LIN {X 0,Y 547.028,Z 596.722,A -85,B 0,C 180,E1 3579.172,E2 3579.172} C_VEL
LIN {X 0,Y 546.524,Z 623.669,A -85,B 0,C 180,E1 3580.328,E2 3580.328} C_VEL
LIN {X 0,Y 545.905,Z 649.048,A -85,B 0,C 180,E1 3582.094,E2 3582.094} C_VEL
LIN {X 0,Y 545.325,Z 670.672,A -85,B 0,C 180,E1 3584.351,E2 3584.351} C_VEL
LIN {X 0,Y 545.02,Z 688.06,A -85,B 0,C 180,E1 3587.017,E2 3587.017} C_VEL
LIN {X 0,Y 544.801,Z 699.894,A -85,B 0,C 180,E1 3589.924,E2 3589.924} C_VEL
LIN {X 0,Y 544.735,Z 704.998,A -85,B 0,C 180,E1 3592.042,E2 3592.042} C_VEL
LIN {X 0,Y 544.721,Z 707.404,A -85,B 0,C 180,E1 3595.236,E2 3595.236} C_VEL
LIN {X 0,Y 544.817,Z 705.335,A -85,B 0,C 180,E1 3597.622,E2 3597.622} C_VEL
LIN {X 0,Y 544.899,Z 697.263,A -85,B 0,C 180,E1 3600.797,E2 3600.797} C_VEL
LIN {X 0,Y 545.082,Z 683.494,A -85,B 0,C 180,E1 3603.697,E2 3603.697} C_VEL
LIN {X 0,Y 545.462,Z 664.993,A -85,B 0,C 180,E1 3606.247,E2 3606.247} C_VEL
LIN {X 0,Y 546.119,Z 641.134,A -85,B 0,C 180,E1 3608.445,E2 3608.445} C_VEL
LIN {X 0,Y 546.671,Z 615.982,A -85,B 0,C 180,E1 3609.983,E2 3609.983} C_VEL
LIN {X 0,Y 547.21,Z 587.354,A -85,B 0,C 180,E1 3611.001,E2 3611.001} C_VEL
LIN {X 0,Y 546.153,Z 557.095,A -85,B 0,C 180,E1 3611.528,E2 3611.528} C_VEL
LIN {X 0,Y 544.539,Z 549.53,A -85,B 0,C 180,E1 3611.757,E2 3611.757} C_VEL
LIN {X 0,Y 544.29,Z 549.53,A -85,B 0,C 180,E1 3617.76,E2 3617.76} C_VEL
LIN {X 0,Y 544.118,Z 549.53,A -85,B 0,C 180,E1 3623.753,E2 3623.753} C_VEL
LIN {X 0,Y 543.994,Z 549.53,A -85,B 0,C 180,E1 3629.959,E2 3629.959} C_VEL
LIN {X 0,Y 543.92,Z 549.53,A -85,B 0,C 180,E1 3635.639,E2 3635.639} C_VEL
LIN {X 0,Y 543.965,Z 549.53,A -85,B 0,C 180,E1 3641.748,E2 3641.748} C_VEL
LIN {X 0,Y 544.059,Z 549.53,A -85,B 0,C 180,E1 3648.261,E2 3648.261} C_VEL
LIN {X 0,Y 543.981,Z 549.53,A -85,B 0,C 180,E1 3654.366,E2 3654.366} C_VEL
LIN {X 0,Y 543.974,Z 549.53,A -85,B 0,C 180,E1 3660.041,E2 3660.041} C_VEL
LIN {X 0,Y 544.383,Z 549.53,A -85,B 0,C 180,E1 3664.815,E2 3664.815} C_VEL
LIN {X 0,Y 551.536,Z 570.193,A -85,B 0,C 180,E1 3665.614,E2 3665.614} C_VEL
LIN {X 0,Y 550.555,Z 607.701,A -85,B 0,C 180,E1 3666.786,E2 3666.786} C_VEL
LIN {X 0,Y 549.229,Z 644.248,A -85,B 0,C 180,E1 3668.649,E2 3668.649} C_VEL
LIN {X 0,Y 547.877,Z 676.541,A -85,B 0,C 180,E1 3670.994,E2 3670.994} C_VEL
LIN {X 0,Y 546.564,Z 706.625,A -85,B 0,C 180,E1 3673.971,E2 3673.971} C_VEL
LIN {X 0,Y 545.565,Z 730.848,A -85,B 0,C 180,E1 3677.215,E2 3677.215} C_VEL
LIN {X 0,Y 545.084,Z 748.889,A -85,B 0,C 180,E1 3680.438,E2 3680.438} C_VEL
LIN {X 0,Y 544.734,Z 763.268,A -85,B 0,C 180,E1 3684.037,E2 3684.037} C_VEL
LIN {X 0,Y 544.715,Z 772.438,A -85,B 0,C 180,E1 3687.618,E2 3687.618} C_VEL
LIN {X 0,Y 544.588,Z 777.144,A -85,B 0,C 180,E1 3691.588,E2 3691.588} C_VEL
LIN {X 0,Y 544.66,Z 776.874,A -85,B 0,C 180,E1 3694.769,E2 3694.769} C_VEL
LIN {X 0,Y 544.677,Z 771.522,A -85,B 0,C 180,E1 3698.766,E2 3698.766} C_VEL
LIN {X 0,Y 544.773,Z 761.522,A -85,B 0,C 180,E1 3702.398,E2 3702.398} C_VEL
LIN {X 0,Y 545.169,Z 745.947,A -85,B 0,C 180,E1 3706.071,E2 3706.071} C_VEL
LIN {X 0,Y 545.847,Z 724.204,A -85,B 0,C 180,E1 3709.682,E2 3709.682} C_VEL
LIN {X 0,Y 546.935,Z 698.541,A -85,B 0,C 180,E1 3712.832,E2 3712.832} C_VEL
LIN {X 0,Y 548.289,Z 666.942,A -85,B 0,C 180,E1 3715.697,E2 3715.697} C_VEL
LIN {X 0,Y 549.53,Z 634.518,A -85,B 0,C 180,E1 3717.832,E2 3717.832} C_VEL
LIN {X 0,Y 550.827,Z 598.514,A -85,B 0,C 180,E1 3719.477,E2 3719.477} C_VEL
LIN {X 0,Y 550.795,Z 568.148,A -85,B 0,C 180,E1 3720.384,E2 3720.384} C_VEL
LIN {X 0,Y 544.129,Z 549.53,A -85,B 0,C 180,E1 3721.134,E2 3721.134} C_VEL
LIN {X 0,Y 544.13,Z 549.53,A -85,B 0,C 180,E1 3726.456,E2 3726.456} C_VEL
LIN {X 0,Y 544.008,Z 549.53,A -85,B 0,C 180,E1 3731.744,E2 3731.744} C_VEL
LIN {X 0,Y 544.033,Z 549.53,A -85,B 0,C 180,E1 3738.504,E2 3738.504} C_VEL
LIN {X 0,Y 544.169,Z 549.53,A -85,B 0,C 180,E1 3744.38,E2 3744.38} C_VEL
LIN {X 0,Y 544.074,Z 549.53,A -85,B 0,C 180,E1 3750.046,E2 3750.046} C_VEL
LIN {X 0,Y 544.017,Z 549.53,A -85,B 0,C 180,E1 3756.273,E2 3756.273} C_VEL
LIN {X 0,Y 544.219,Z 549.53,A -85,B 0,C 180,E1 3761.604,E2 3761.604} C_VEL
LIN {X 0,Y 546.614,Z 578.067,A -85,B 0,C 180,E1 3762.063,E2 3762.063} C_VEL
LIN {X 0,Y 546.452,Z 611.547,A -85,B 0,C 180,E1 3762.642,E2 3762.642} C_VEL
LIN {X 0,Y 546.062,Z 638.227,A -85,B 0,C 180,E1 3763.751,E2 3763.751} C_VEL
LIN {X 0,Y 545.544,Z 661.449,A -85,B 0,C 180,E1 3765.432,E2 3765.432} C_VEL
LIN {X 0,Y 545.125,Z 679.302,A -85,B 0,C 180,E1 3767.405,E2 3767.405} C_VEL
LIN {X 0,Y 544.917,Z 694.025,A -85,B 0,C 180,E1 3769.891,E2 3769.891} C_VEL
LIN {X 0,Y 544.794,Z 703.355,A -85,B 0,C 180,E1 3772.538,E2 3772.538} C_VEL
LIN {X 0,Y 544.727,Z 707.246,A -85,B 0,C 180,E1 3775.229,E2 3775.229} C_VEL
LIN {X 0,Y 544.711,Z 707.192,A -85,B 0,C 180,E1 3776.82,E2 3776.82} C_VEL
LIN {X 0,Y 544.857,Z 702.766,A -85,B 0,C 180,E1 3779.6,E2 3779.6} C_VEL
LIN {X 0,Y 544.936,Z 692.366,A -85,B 0,C 180,E1 3782.377,E2 3782.377} C_VEL
LIN {X 0,Y 545.244,Z 676.093,A -85,B 0,C 180,E1 3784.92,E2 3784.92} C_VEL
LIN {X 0,Y 545.685,Z 656.173,A -85,B 0,C 180,E1 3786.945,E2 3786.945} C_VEL
LIN {X 0,Y 546.186,Z 633.014,A -85,B 0,C 180,E1 3788.436,E2 3788.436} C_VEL
LIN {X 0,Y 546.479,Z 607.222,A -85,B 0,C 180,E1 3789.383,E2 3789.383} C_VEL
LIN {X 0,Y 545.692,Z 554.823,A -85,B 0,C 180,E1 3790.17,E2 3790.17} C_VEL
LIN {X 0,Y 544.581,Z 549.53,A -85,B 0,C 180,E1 3790.348,E2 3790.348} C_VEL
LIN {X 0,Y 544.209,Z 549.53,A -85,B 0,C 180,E1 3792.982,E2 3792.982} C_VEL
LIN {X 0,Y 540.252,Z 549.53,A -85,B 0,C 180,E1 3794.779,E2 3794.779} C_VEL
LIN {X 0,Y 536.278,Z 549.53,A -85,B 0,C 180,E1 3796.602,E2 3796.602} C_VEL
LIN {X 0,Y 536.17,Z 549.53,A -85,B 0,C 180,E1 3801.741,E2 3801.741} C_VEL
LIN {X 0,Y 536.063,Z 549.53,A -85,B 0,C 180,E1 3806.765,E2 3806.765} C_VEL
LIN {X 0,Y 535.986,Z 549.53,A -85,B 0,C 180,E1 3812.358,E2 3812.358} C_VEL
LIN {X 0,Y 536.152,Z 549.53,A -85,B 0,C 180,E1 3818.253,E2 3818.253} C_VEL
LIN {X 0,Y 536.007,Z 549.53,A -85,B 0,C 180,E1 3824.73,E2 3824.73} C_VEL
LIN {X 0,Y 535.97,Z 549.53,A -85,B 0,C 180,E1 3829.636,E2 3829.636} C_VEL
LIN {X 0,Y 536.088,Z 550.016,A -85,B 0,C 180,E1 3835.356,E2 3835.356} C_VEL
LIN {X 0,Y 537.029,Z 553.098,A -85,B 0,C 180,E1 3836.078,E2 3836.078} C_VEL
LIN {X 0,Y 547.19,Z 573.958,A -85,B 0,C 180,E1 3837.11,E2 3837.11} C_VEL
LIN {X 0,Y 546.77,Z 626.968,A -85,B 0,C 180,E1 3838.085,E2 3838.085} C_VEL
LIN {X 0,Y 545.503,Z 664.523,A -85,B 0,C 180,E1 3839.384,E2 3839.384} C_VEL
LIN {X 0,Y 543.745,Z 701.396,A -85,B 0,C 180,E1 3841.3,E2 3841.3} C_VEL
LIN {X 0,Y 541.756,Z 736.91,A -85,B 0,C 180,E1 3843.864,E2 3843.864} C_VEL
LIN {X 0,Y 539.937,Z 768.966,A -85,B 0,C 180,E1 3846.963,E2 3846.963} C_VEL
LIN {X 0,Y 538.457,Z 797.181,A -85,B 0,C 180,E1 3850.559,E2 3850.559} C_VEL
LIN {X 0,Y 537.455,Z 819.461,A -85,B 0,C 180,E1 3854.319,E2 3854.319} C_VEL
LIN {X 0,Y 536.952,Z 836.542,A -85,B 0,C 180,E1 3858.242,E2 3858.242} C_VEL
LIN {X 0,Y 536.771,Z 847.704,A -85,B 0,C 180,E1 3861.918,E2 3861.918} C_VEL
LIN {X 0,Y 536.661,Z 853.979,A -85,B 0,C 180,E1 3865.16,E2 3865.16} C_VEL
LIN {X 0,Y 536.666,Z 857.105,A -85,B 0,C 180,E1 3868.388,E2 3868.388} C_VEL
LIN {X 0,Y 536.801,Z 857.105,A -85,B 0,C 180,E1 3871.611,E2 3871.611} C_VEL
LIN {X 0,Y 536.76,Z 852.747,A -85,B 0,C 180,E1 3875.647,E2 3875.647} C_VEL
LIN {X 0,Y 536.826,Z 843.325,A -85,B 0,C 180,E1 3879.711,E2 3879.711} C_VEL
LIN {X 0,Y 537.257,Z 827.755,A -85,B 0,C 180,E1 3883.938,E2 3883.938} C_VEL
LIN {X 0,Y 538.05,Z 806.656,A -85,B 0,C 180,E1 3887.971,E2 3887.971} C_VEL
LIN {X 0,Y 539.341,Z 780.531,A -85,B 0,C 180,E1 3891.684,E2 3891.684} C_VEL
LIN {X 0,Y 541.056,Z 749.2,A -85,B 0,C 180,E1 3895.049,E2 3895.049} C_VEL
LIN {X 0,Y 543.025,Z 714.333,A -85,B 0,C 180,E1 3897.86,E2 3897.86} C_VEL
LIN {X 0,Y 544.929,Z 676.974,A -85,B 0,C 180,E1 3900.05,E2 3900.05} C_VEL
LIN {X 0,Y 546.442,Z 637.3,A -85,B 0,C 180,E1 3901.622,E2 3901.622} C_VEL
LIN {X 0,Y 547.443,Z 597.917,A -85,B 0,C 180,E1 3902.505,E2 3902.505} C_VEL
LIN {X 0,Y 546.759,Z 573.274,A -85,B 0,C 180,E1 3902.929,E2 3902.929} C_VEL
LIN {X 0,Y 536.066,Z 549.77,A -85,B 0,C 180,E1 3904.094,E2 3904.094} C_VEL
LIN {X 0,Y 536.186,Z 549.53,A -85,B 0,C 180,E1 3908.259,E2 3908.259} C_VEL
LIN {X 0,Y 535.987,Z 549.53,A -85,B 0,C 180,E1 3914.742,E2 3914.742} C_VEL
LIN {X 0,Y 536.086,Z 549.53,A -85,B 0,C 180,E1 3919.657,E2 3919.657} C_VEL
LIN {X 0,Y 536.037,Z 549.53,A -85,B 0,C 180,E1 3924.733,E2 3924.733} C_VEL
LIN {X 0,Y 536.049,Z 549.53,A -85,B 0,C 180,E1 3930.781,E2 3930.781} C_VEL
LIN {X 0,Y 536.168,Z 549.53,A -85,B 0,C 180,E1 3936.799,E2 3936.799} C_VEL
LIN {X 0,Y 536.352,Z 549.882,A -85,B 0,C 180,E1 3938.06,E2 3938.06} C_VEL
LIN {X 0,Y 539.4,Z 567.141,A -85,B 0,C 180,E1 3938.367,E2 3938.367} C_VEL
LIN {X 0,Y 539.351,Z 599.199,A -85,B 0,C 180,E1 3939.037,E2 3939.037} C_VEL
LIN {X 0,Y 538.815,Z 627.007,A -85,B 0,C 180,E1 3940.276,E2 3940.276} C_VEL
LIN {X 0,Y 538.193,Z 651.43,A -85,B 0,C 180,E1 3942.039,E2 3942.039} C_VEL
LIN {X 0,Y 537.578,Z 672.435,A -85,B 0,C 180,E1 3944.329,E2 3944.329} C_VEL
LIN {X 0,Y 537.147,Z 688.92,A -85,B 0,C 180,E1 3947.016,E2 3947.016} C_VEL
LIN {X 0,Y 536.867,Z 701.196,A -85,B 0,C 180,E1 3950.294,E2 3950.294} C_VEL
LIN {X 0,Y 536.836,Z 704.882,A -85,B 0,C 180,E1 3951.924,E2 3951.924} C_VEL
LIN {X 0,Y 536.812,Z 707.4,A -85,B 0,C 180,E1 3955.166,E2 3955.166} C_VEL
LIN {X 0,Y 536.855,Z 704.123,A -85,B 0,C 180,E1 3958.393,E2 3958.393} C_VEL
LIN {X 0,Y 536.903,Z 694.456,A -85,B 0,C 180,E1 3961.614,E2 3961.614} C_VEL
LIN {X 0,Y 537.262,Z 681.227,A -85,B 0,C 180,E1 3964.279,E2 3964.279} C_VEL
LIN {X 0,Y 537.883,Z 661.608,A -85,B 0,C 180,E1 3966.852,E2 3966.852} C_VEL
LIN {X 0,Y 538.498,Z 638.728,A -85,B 0,C 180,E1 3968.87,E2 3968.87} C_VEL
LIN {X 0,Y 539.16,Z 612.131,A -85,B 0,C 180,E1 3970.384,E2 3970.384} C_VEL
LIN {X 0,Y 539.616,Z 584.105,A -85,B 0,C 180,E1 3971.293,E2 3971.293} C_VEL
LIN {X 0,Y 538.584,Z 558.624,A -85,B 0,C 180,E1 3971.715,E2 3971.715} C_VEL
LIN {X 0,Y 536.63,Z 549.53,A -85,B 0,C 180,E1 3971.902,E2 3971.902} C_VEL
LIN {X 0,Y 536.36,Z 549.53,A -85,B 0,C 180,E1 3978.032,E2 3978.032} C_VEL
LIN {X 0,Y 536.24,Z 549.53,A -85,B 0,C 180,E1 3983.206,E2 3983.206} C_VEL
LIN {X 0,Y 536.062,Z 549.53,A -85,B 0,C 180,E1 3989.221,E2 3989.221} C_VEL
LIN {X 0,Y 536.025,Z 549.53,A -85,B 0,C 180,E1 3994.271,E2 3994.271} C_VEL
LIN {X 0,Y 535.971,Z 549.53,A -85,B 0,C 180,E1 4000.513,E2 4000.513} C_VEL
LIN {X 0,Y 536.049,Z 549.53,A -85,B 0,C 180,E1 4007.053,E2 4007.053} C_VEL
LIN {X 0,Y 536.15,Z 549.53,A -85,B 0,C 180,E1 4012.012,E2 4012.012} C_VEL
LIN {X 0,Y 536.009,Z 549.53,A -85,B 0,C 180,E1 4017.659,E2 4017.659} C_VEL
LIN {X 0,Y 536.434,Z 549.53,A -85,B 0,C 180,E1 4024.363,E2 4024.363} C_VEL
LIN {X 0,Y 544.5,Z 571.697,A -85,B 0,C 180,E1 4025.269,E2 4025.269} C_VEL
LIN {X 0,Y 543.373,Z 608.888,A -85,B 0,C 180,E1 4026.466,E2 4026.466} C_VEL
LIN {X 0,Y 541.907,Z 644.984,A -85,B 0,C 180,E1 4028.346,E2 4028.346} C_VEL
LIN {X 0,Y 540.436,Z 676.308,A -85,B 0,C 180,E1 4030.655,E2 4030.655} C_VEL
LIN {X 0,Y 538.983,Z 705.238,A -85,B 0,C 180,E1 4033.531,E2 4033.531} C_VEL
LIN {X 0,Y 537.85,Z 729.819,A -85,B 0,C 180,E1 4036.822,E2 4036.822} C_VEL
LIN {X 0,Y 537.262,Z 749.105,A -85,B 0,C 180,E1 4040.297,E2 4040.297} C_VEL
LIN {X 0,Y 536.857,Z 763.401,A -85,B 0,C 180,E1 4043.949,E2 4043.949} C_VEL
LIN {X 0,Y 536.833,Z 772.522,A -85,B 0,C 180,E1 4047.583,E2 4047.583} C_VEL
LIN {X 0,Y 536.698,Z 777.155,A -85,B 0,C 180,E1 4051.612,E2 4051.612} C_VEL
LIN {X 0,Y 536.752,Z 776.846,A -85,B 0,C 180,E1 4054.839,E2 4054.839} C_VEL
LIN {X 0,Y 536.791,Z 771.439,A -85,B 0,C 180,E1 4058.896,E2 4058.896} C_VEL
LIN {X 0,Y 536.909,Z 761.358,A -85,B 0,C 180,E1 4062.583,E2 4062.583} C_VEL
LIN {X 0,Y 537.478,Z 744.404,A -85,B 0,C 180,E1 4066.568,E2 4066.568} C_VEL
LIN {X 0,Y 538.324,Z 721.745,A -85,B 0,C 180,E1 4070.279,E2 4070.279} C_VEL
LIN {X 0,Y 539.492,Z 694.967,A -85,B 0,C 180,E1 4073.493,E2 4073.493} C_VEL
LIN {X 0,Y 540.953,Z 665.008,A -85,B 0,C 180,E1 4076.177,E2 4076.177} C_VEL
LIN {X 0,Y 542.504,Z 629.524,A -85,B 0,C 180,E1 4078.465,E2 4078.465} C_VEL
LIN {X 0,Y 543.811,Z 593.165,A -85,B 0,C 180,E1 4080.033,E2 4080.033} C_VEL
LIN {X 0,Y 543.789,Z 570.399,A -85,B 0,C 180,E1 4080.716,E2 4080.716} C_VEL
LIN {X 0,Y 536.243,Z 549.53,A -85,B 0,C 180,E1 4081.594,E2 4081.594} C_VEL
LIN {X 0,Y 536.225,Z 549.53,A -85,B 0,C 180,E1 4086.231,E2 4086.231} C_VEL
LIN {X 0,Y 535.988,Z 549.53,A -85,B 0,C 180,E1 4092.514,E2 4092.514} C_VEL
LIN {X 0,Y 536.002,Z 549.53,A -85,B 0,C 180,E1 4097.488,E2 4097.488} C_VEL
LIN {X 0,Y 536.248,Z 549.53,A -85,B 0,C 180,E1 4103.771,E2 4103.771} C_VEL
LIN {X 0,Y 536.183,Z 549.53,A -85,B 0,C 180,E1 4109.559,E2 4109.559} C_VEL
LIN {X 0,Y 536.048,Z 549.53,A -85,B 0,C 180,E1 4115.018,E2 4115.018} C_VEL
LIN {X 0,Y 536.304,Z 549.53,A -85,B 0,C 180,E1 4121.416,E2 4121.416} C_VEL
LIN {X 0,Y 538.926,Z 577.898,A -85,B 0,C 180,E1 4121.874,E2 4121.874} C_VEL
LIN {X 0,Y 538.796,Z 613.16,A -85,B 0,C 180,E1 4122.493,E2 4122.493} C_VEL
LIN {X 0,Y 538.407,Z 638.091,A -85,B 0,C 180,E1 4123.531,E2 4123.531} C_VEL
LIN {X 0,Y 537.887,Z 661.122,A -85,B 0,C 180,E1 4125.163,E2 4125.163} C_VEL
LIN {X 0,Y 537.428,Z 679.88,A -85,B 0,C 180,E1 4127.221,E2 4127.221} C_VEL
LIN {X 0,Y 537.121,Z 694.712,A -85,B 0,C 180,E1 4129.759,E2 4129.759} C_VEL
LIN {X 0,Y 536.956,Z 704.116,A -85,B 0,C 180,E1 4132.536,E2 4132.536} C_VEL
LIN {X 0,Y 536.848,Z 707.814,A -85,B 0,C 180,E1 4135.159,E2 4135.159} C_VEL
LIN {X 0,Y 536.839,Z 707.82,A -85,B 0,C 180,E1 4136.773,E2 4136.773} C_VEL
LIN {X 0,Y 537.025,Z 703.659,A -85,B 0,C 180,E1 4139.594,E2 4139.594} C_VEL
LIN {X 0,Y 537.169,Z 693.667,A -85,B 0,C 180,E1 4142.411,E2 4142.411} C_VEL
LIN {X 0,Y 537.499,Z 679.034,A -85,B 0,C 180,E1 4144.828,E2 4144.828} C_VEL
LIN {X 0,Y 537.97,Z 659.107,A -85,B 0,C 180,E1 4146.944,E2 4146.944} C_VEL
LIN {X 0,Y 538.485,Z 636.872,A -85,B 0,C 180,E1 4148.457,E2 4148.457} C_VEL
LIN {X 0,Y 538.755,Z 611.43,A -85,B 0,C 180,E1 4149.468,E2 4149.468} C_VEL
LIN {X 0,Y 537.977,Z 556.066,A -85,B 0,C 180,E1 4150.34,E2 4150.34} C_VEL
LIN {X 0,Y 536.672,Z 549.53,A -85,B 0,C 180,E1 4150.504,E2 4150.504} C_VEL
LIN {X 0,Y 536.278,Z 549.53,A -85,B 0,C 180,E1 4156.602,E2 4156.602} C_VEL
LIN {X 0,Y 532.315,Z 549.53,A -85,B 0,C 180,E1 4158.428,E2 4158.428} C_VEL
LIN {X 0,Y 528.28,Z 549.53,A -85,B 0,C 180,E1 4160.281,E2 4160.281} C_VEL
LIN {X 0,Y 528.189,Z 549.53,A -85,B 0,C 180,E1 4165.371,E2 4165.371} C_VEL
LIN {X 0,Y 528.066,Z 549.53,A -85,B 0,C 180,E1 4170.976,E2 4170.976} C_VEL
LIN {X 0,Y 528.175,Z 549.53,A -85,B 0,C 180,E1 4176.864,E2 4176.864} C_VEL
LIN {X 0,Y 528.11,Z 549.53,A -85,B 0,C 180,E1 4183.292,E2 4183.292} C_VEL
LIN {X 0,Y 528.004,Z 549.53,A -85,B 0,C 180,E1 4188.898,E2 4188.898} C_VEL
LIN {X 0,Y 528.138,Z 550.181,A -85,B 0,C 180,E1 4194.065,E2 4194.065} C_VEL
LIN {X 0,Y 531.093,Z 555.687,A -85,B 0,C 180,E1 4194.979,E2 4194.979} C_VEL
LIN {X 0,Y 533.002,Z 560.67,A -85,B 0,C 180,E1 4195.907,E2 4195.907} C_VEL
LIN {X 0,Y 540.709,Z 578.275,A -85,B 0,C 180,E1 4196.732,E2 4196.732} C_VEL
LIN {X 0,Y 540.02,Z 627.687,A -85,B 0,C 180,E1 4197.659,E2 4197.659} C_VEL
LIN {X 0,Y 538.569,Z 666.039,A -85,B 0,C 180,E1 4199.016,E2 4199.016} C_VEL
LIN {X 0,Y 536.615,Z 702.707,A -85,B 0,C 180,E1 4200.969,E2 4200.969} C_VEL
LIN {X 0,Y 534.413,Z 738.192,A -85,B 0,C 180,E1 4203.591,E2 4203.591} C_VEL
LIN {X 0,Y 532.345,Z 770.593,A -85,B 0,C 180,E1 4206.804,E2 4206.804} C_VEL
LIN {X 0,Y 530.709,Z 798.609,A -85,B 0,C 180,E1 4210.48,E2 4210.48} C_VEL
LIN {X 0,Y 529.619,Z 821.558,A -85,B 0,C 180,E1 4214.505,E2 4214.505} C_VEL
LIN {X 0,Y 529.072,Z 838.032,A -85,B 0,C 180,E1 4218.482,E2 4218.482} C_VEL
LIN {X 0,Y 528.912,Z 849.601,A -85,B 0,C 180,E1 4222.622,E2 4222.622} C_VEL
LIN {X 0,Y 528.783,Z 855.935,A -85,B 0,C 180,E1 4226.727,E2 4226.727} C_VEL
LIN {X 0,Y 528.794,Z 857.5,A -85,B 0,C 180,E1 4230,E2 4230} C_VEL
LIN {X 0,Y 528.777,Z 855.936,A -85,B 0,C 180,E1 4233.272,E2 4233.272} C_VEL
LIN {X 0,Y 528.902,Z 849.602,A -85,B 0,C 180,E1 4237.377,E2 4237.377} C_VEL
LIN {X 0,Y 529.092,Z 838.035,A -85,B 0,C 180,E1 4241.517,E2 4241.517} C_VEL
LIN {X 0,Y 529.756,Z 820.519,A -85,B 0,C 180,E1 4245.702,E2 4245.702} C_VEL
LIN {X 0,Y 530.846,Z 797.184,A -85,B 0,C 180,E1 4249.731,E2 4249.731} C_VEL
LIN {X 0,Y 532.525,Z 768.976,A -85,B 0,C 180,E1 4253.376,E2 4253.376} C_VEL
LIN {X 0,Y 534.454,Z 737.299,A -85,B 0,C 180,E1 4256.486,E2 4256.486} C_VEL
LIN {X 0,Y 536.65,Z 701.465,A -85,B 0,C 180,E1 4259.111,E2 4259.111} C_VEL
LIN {X 0,Y 538.616,Z 663.303,A -85,B 0,C 180,E1 4261.106,E2 4261.106} C_VEL
LIN {X 0,Y 540.13,Z 624.026,A -85,B 0,C 180,E1 4262.435,E2 4262.435} C_VEL
LIN {X 0,Y 540.1,Z 575.719,A -85,B 0,C 180,E1 4263.35,E2 4263.35} C_VEL
LIN {X 0,Y 531.834,Z 558.071,A -85,B 0,C 180,E1 4264.291,E2 4264.291} C_VEL
LIN {X 0,Y 528.419,Z 551.415,A -85,B 0,C 180,E1 4265.476,E2 4265.476} C_VEL
LIN {X 0,Y 528.198,Z 549.53,A -85,B 0,C 180,E1 4265.835,E2 4265.835} C_VEL
LIN {X 0,Y 528.061,Z 549.53,A -85,B 0,C 180,E1 4271.096,E2 4271.096} C_VEL
LIN {X 0,Y 528.106,Z 549.53,A -85,B 0,C 180,E1 4276.708,E2 4276.708} C_VEL
LIN {X 0,Y 528.193,Z 549.53,A -85,B 0,C 180,E1 4283.137,E2 4283.137} C_VEL
LIN {X 0,Y 528.139,Z 549.53,A -85,B 0,C 180,E1 4289.053,E2 4289.053} C_VEL
LIN {X 0,Y 528.245,Z 549.53,A -85,B 0,C 180,E1 4294.632,E2 4294.632} C_VEL
LIN {X 0,Y 528.402,Z 549.53,A -85,B 0,C 180,E1 4297.823,E2 4297.823} C_VEL
LIN {X 0,Y 531.722,Z 567.317,A -85,B 0,C 180,E1 4298.177,E2 4298.177} C_VEL
LIN {X 0,Y 531.703,Z 599.569,A -85,B 0,C 180,E1 4298.836,E2 4298.836} C_VEL
LIN {X 0,Y 531.19,Z 627.675,A -85,B 0,C 180,E1 4300.072,E2 4300.072} C_VEL
LIN {X 0,Y 530.543,Z 652.655,A -85,B 0,C 180,E1 4301.883,E2 4301.883} C_VEL
LIN {X 0,Y 529.918,Z 673.058,A -85,B 0,C 180,E1 4304.096,E2 4304.096} C_VEL
LIN {X 0,Y 529.459,Z 689.802,A -85,B 0,C 180,E1 4306.824,E2 4306.824} C_VEL
LIN {X 0,Y 529.163,Z 700.398,A -85,B 0,C 180,E1 4309.518,E2 4309.518} C_VEL
LIN {X 0,Y 528.974,Z 706.925,A -85,B 0,C 180,E1 4312.628,E2 4312.628} C_VEL
LIN {X 0,Y 528.987,Z 708.319,A -85,B 0,C 180,E1 4315.094,E2 4315.094} C_VEL
LIN {X 0,Y 529.036,Z 705.204,A -85,B 0,C 180,E1 4318.369,E2 4318.369} C_VEL
LIN {X 0,Y 529.149,Z 695.94,A -85,B 0,C 180,E1 4321.638,E2 4321.638} C_VEL
LIN {X 0,Y 529.562,Z 681.735,A -85,B 0,C 180,E1 4324.498,E2 4324.498} C_VEL
LIN {X 0,Y 530.195,Z 663.169,A -85,B 0,C 180,E1 4326.951,E2 4326.951} C_VEL
LIN {X 0,Y 530.82,Z 640.298,A -85,B 0,C 180,E1 4328.999,E2 4328.999} C_VEL
LIN {X 0,Y 531.538,Z 613.974,A -85,B 0,C 180,E1 4330.535,E2 4330.535} C_VEL
LIN {X 0,Y 531.99,Z 586.512,A -85,B 0,C 180,E1 4331.457,E2 4331.457} C_VEL
LIN {X 0,Y 530.973,Z 559.89,A -85,B 0,C 180,E1 4331.912,E2 4331.912} C_VEL
LIN {X 0,Y 528.741,Z 549.53,A -85,B 0,C 180,E1 4332.126,E2 4332.126} C_VEL
LIN {X 0,Y 528.427,Z 549.53,A -85,B 0,C 180,E1 4338.312,E2 4338.312} C_VEL
LIN {X 0,Y 528.258,Z 549.53,A -85,B 0,C 180,E1 4343.907,E2 4343.907} C_VEL
LIN {X 0,Y 528.196,Z 549.53,A -85,B 0,C 180,E1 4349.061,E2 4349.061} C_VEL
LIN {X 0,Y 528.089,Z 549.53,A -85,B 0,C 180,E1 4354.86,E2 4354.86} C_VEL
LIN {X 0,Y 528.01,Z 549.53,A -85,B 0,C 180,E1 4361.101,E2 4361.101} C_VEL
LIN {X 0,Y 528.099,Z 549.53,A -85,B 0,C 180,E1 4366.697,E2 4366.697} C_VEL
LIN {X 0,Y 528.172,Z 549.53,A -85,B 0,C 180,E1 4373.135,E2 4373.135} C_VEL
LIN {X 0,Y 528.093,Z 549.53,A -85,B 0,C 180,E1 4379.043,E2 4379.043} C_VEL
LIN {X 0,Y 528.418,Z 549.53,A -85,B 0,C 180,E1 4383.898,E2 4383.898} C_VEL
LIN {X 0,Y 537.464,Z 574.695,A -85,B 0,C 180,E1 4384.952,E2 4384.952} C_VEL
LIN {X 0,Y 536.224,Z 609.88,A -85,B 0,C 180,E1 4386.131,E2 4386.131} C_VEL
LIN {X 0,Y 534.613,Z 645.72,A -85,B 0,C 180,E1 4388.035,E2 4388.035} C_VEL
LIN {X 0,Y 532.907,Z 677.756,A -85,B 0,C 180,E1 4390.457,E2 4390.457} C_VEL
LIN {X 0,Y 531.281,Z 707.393,A -85,B 0,C 180,E1 4393.497,E2 4393.497} C_VEL
LIN {X 0,Y 529.985,Z 732.738,A -85,B 0,C 180,E1 4397.042,E2 4397.042} C_VEL
LIN {X 0,Y 529.351,Z 751.16,A -85,B 0,C 180,E1 4400.565,E2 4400.565} C_VEL
LIN {X 0,Y 528.95,Z 764.807,A -85,B 0,C 180,E1 4404.269,E2 4404.269} C_VEL
LIN {X 0,Y 528.94,Z 772.598,A -85,B 0,C 180,E1 4407.543,E2 4407.543} C_VEL
LIN {X 0,Y 528.796,Z 777.166,A -85,B 0,C 180,E1 4411.636,E2 4411.636} C_VEL
LIN {X 0,Y 528.871,Z 776.811,A -85,B 0,C 180,E1 4414.911,E2 4414.911} C_VEL
LIN {X 0,Y 528.893,Z 771.356,A -85,B 0,C 180,E1 4419.03,E2 4419.03} C_VEL
LIN {X 0,Y 529.05,Z 761.194,A -85,B 0,C 180,E1 4422.773,E2 4422.773} C_VEL
LIN {X 0,Y 529.678,Z 744.327,A -85,B 0,C 180,E1 4426.788,E2 4426.788} C_VEL
LIN {X 0,Y 530.591,Z 722.579,A -85,B 0,C 180,E1 4430.417,E2 4430.417} C_VEL
LIN {X 0,Y 531.826,Z 696.836,A -85,B 0,C 180,E1 4433.602,E2 4433.602} C_VEL
LIN {X 0,Y 533.541,Z 665.8,A -85,B 0,C 180,E1 4436.456,E2 4436.456} C_VEL
LIN {X 0,Y 535.191,Z 631.448,A -85,B 0,C 180,E1 4438.725,E2 4438.725} C_VEL
LIN {X 0,Y 536.701,Z 595.377,A -85,B 0,C 180,E1 4440.343,E2 4440.343} C_VEL
LIN {X 0,Y 536.756,Z 572.463,A -85,B 0,C 180,E1 4441.064,E2 4441.064} C_VEL
LIN {X 0,Y 528.375,Z 549.53,A -85,B 0,C 180,E1 4442.055,E2 4442.055} C_VEL
LIN {X 0,Y 528.258,Z 549.53,A -85,B 0,C 180,E1 4446.878,E2 4446.878} C_VEL
LIN {X 0,Y 528.01,Z 549.53,A -85,B 0,C 180,E1 4453.313,E2 4453.313} C_VEL
LIN {X 0,Y 528.085,Z 549.53,A -85,B 0,C 180,E1 4458.906,E2 4458.906} C_VEL
LIN {X 0,Y 528.345,Z 549.53,A -85,B 0,C 180,E1 4465.16,E2 4465.16} C_VEL
LIN {X 0,Y 528.203,Z 549.53,A -85,B 0,C 180,E1 4470.939,E2 4470.939} C_VEL
LIN {X 0,Y 528.162,Z 549.53,A -85,B 0,C 180,E1 4476.418,E2 4476.418} C_VEL
LIN {X 0,Y 528.369,Z 549.563,A -85,B 0,C 180,E1 4481.215,E2 4481.215} C_VEL
LIN {X 0,Y 531.256,Z 577.767,A -85,B 0,C 180,E1 4481.681,E2 4481.681} C_VEL
LIN {X 0,Y 531.088,Z 614.753,A -85,B 0,C 180,E1 4482.339,E2 4482.339} C_VEL
LIN {X 0,Y 530.7,Z 639.484,A -85,B 0,C 180,E1 4483.391,E2 4483.391} C_VEL
LIN {X 0,Y 530.164,Z 662.518,A -85,B 0,C 180,E1 4485.048,E2 4485.048} C_VEL
LIN {X 0,Y 529.637,Z 682.007,A -85,B 0,C 180,E1 4487.24,E2 4487.24} C_VEL
LIN {X 0,Y 529.358,Z 696.335,A -85,B 0,C 180,E1 4489.768,E2 4489.768} C_VEL
LIN {X 0,Y 529.166,Z 705.678,A -85,B 0,C 180,E1 4492.623,E2 4492.623} C_VEL
LIN {X 0,Y 529.075,Z 709.089,A -85,B 0,C 180,E1 4495.088,E2 4495.088} C_VEL
LIN {X 0,Y 529.079,Z 709.176,A -85,B 0,C 180,E1 4496.726,E2 4496.726} C_VEL
LIN {X 0,Y 529.199,Z 706.045,A -85,B 0,C 180,E1 4499.179,E2 4499.179} C_VEL
LIN {X 0,Y 529.399,Z 697.05,A -85,B 0,C 180,E1 4502.038,E2 4502.038} C_VEL
LIN {X 0,Y 529.742,Z 682.179,A -85,B 0,C 180,E1 4504.693,E2 4504.693} C_VEL
LIN {X 0,Y 530.237,Z 663.157,A -85,B 0,C 180,E1 4506.841,E2 4506.841} C_VEL
LIN {X 0,Y 530.74,Z 640.534,A -85,B 0,C 180,E1 4508.478,E2 4508.478} C_VEL
LIN {X 0,Y 531.087,Z 615.266,A -85,B 0,C 180,E1 4509.554,E2 4509.554} C_VEL
LIN {X 0,Y 531.144,Z 573.9,A -85,B 0,C 180,E1 4510.266,E2 4510.266} C_VEL
LIN {X 0,Y 530.057,Z 556.125,A -85,B 0,C 180,E1 4510.537,E2 4510.537} C_VEL
LIN {X 0,Y 528.714,Z 549.53,A -85,B 0,C 180,E1 4510.703,E2 4510.703} C_VEL
LIN {X 0,Y 528.401,Z 549.53,A -85,B 0,C 180,E1 4516.59,E2 4516.59} C_VEL
LIN {X 0,Y 528.28,Z 549.53,A -85,B 0,C 180,E1 4520.281,E2 4520.281} C_VEL
LIN {X 0,Y 524.308,Z 549.53,A -85,B 0,C 180,E1 4522.133,E2 4522.133} C_VEL
LIN {X 0,Y 520.273,Z 549.53,A -85,B 0,C 180,E1 4524.012,E2 4524.012} C_VEL
LIN {X 0,Y 520.153,Z 549.53,A -85,B 0,C 180,E1 4529.546,E2 4529.546} C_VEL
LIN {X 0,Y 520.134,Z 549.53,A -85,B 0,C 180,E1 4535.666,E2 4535.666} C_VEL
LIN {X 0,Y 520.214,Z 549.53,A -85,B 0,C 180,E1 4541.037,E2 4541.037} C_VEL
LIN {X 0,Y 520.118,Z 549.53,A -85,B 0,C 180,E1 4546.491,E2 4546.491} C_VEL
LIN {X 0,Y 520.14,Z 549.53,A -85,B 0,C 180,E1 4552.966,E2 4552.966} C_VEL
LIN {X 0,Y 520.219,Z 549.652,A -85,B 0,C 180,E1 4553.486,E2 4553.486} C_VEL
LIN {X 0,Y 523.839,Z 559.232,A -85,B 0,C 180,E1 4554.447,E2 4554.447} C_VEL
LIN {X 0,Y 527.851,Z 565.967,A -85,B 0,C 180,E1 4555.582,E2 4555.582} C_VEL
LIN {X 0,Y 534.116,Z 579.688,A -85,B 0,C 180,E1 4556.29,E2 4556.29} C_VEL
LIN {X 0,Y 533.342,Z 627.768,A -85,B 0,C 180,E1 4557.205,E2 4557.205} C_VEL
LIN {X 0,Y 531.77,Z 665.754,A -85,B 0,C 180,E1 4558.562,E2 4558.562} C_VEL
LIN {X 0,Y 529.596,Z 702.701,A -85,B 0,C 180,E1 4560.546,E2 4560.546} C_VEL
LIN {X 0,Y 527.151,Z 738.185,A -85,B 0,C 180,E1 4563.198,E2 4563.198} C_VEL
LIN {X 0,Y 525.001,Z 768.974,A -85,B 0,C 180,E1 4566.268,E2 4566.268} C_VEL
LIN {X 0,Y 523.15,Z 797.18,A -85,B 0,C 180,E1 4569.966,E2 4569.966} C_VEL
LIN {X 0,Y 521.86,Z 819.459,A -85,B 0,C 180,E1 4573.838,E2 4573.838} C_VEL
LIN {X 0,Y 521.239,Z 836.549,A -85,B 0,C 180,E1 4577.882,E2 4577.882} C_VEL
LIN {X 0,Y 521.012,Z 847.711,A -85,B 0,C 180,E1 4581.672,E2 4581.672} C_VEL
LIN {X 0,Y 520.894,Z 853.984,A -85,B 0,C 180,E1 4585.013,E2 4585.013} C_VEL
LIN {X 0,Y 520.877,Z 857.109,A -85,B 0,C 180,E1 4588.339,E2 4588.339} C_VEL
LIN {X 0,Y 520.999,Z 857.109,A -85,B 0,C 180,E1 4591.66,E2 4591.66} C_VEL
LIN {X 0,Y 520.996,Z 852.745,A -85,B 0,C 180,E1 4595.819,E2 4595.819} C_VEL
LIN {X 0,Y 521.066,Z 843.138,A -85,B 0,C 180,E1 4600.072,E2 4600.072} C_VEL
LIN {X 0,Y 521.644,Z 827.732,A -85,B 0,C 180,E1 4604.369,E2 4604.369} C_VEL
LIN {X 0,Y 522.632,Z 806.653,A -85,B 0,C 180,E1 4608.52,E2 4608.52} C_VEL
LIN {X 0,Y 524.287,Z 780.239,A -85,B 0,C 180,E1 4612.377,E2 4612.377} C_VEL
LIN {X 0,Y 526.4,Z 749.06,A -85,B 0,C 180,E1 4615.812,E2 4615.812} C_VEL
LIN {X 0,Y 528.804,Z 713.987,A -85,B 0,C 180,E1 4618.704,E2 4618.704} C_VEL
LIN {X 0,Y 531.148,Z 676.431,A -85,B 0,C 180,E1 4620.941,E2 4620.941} C_VEL
LIN {X 0,Y 532.952,Z 636.349,A -85,B 0,C 180,E1 4622.549,E2 4622.549} C_VEL
LIN {X 0,Y 534.17,Z 595.742,A -85,B 0,C 180,E1 4623.453,E2 4623.453} C_VEL
LIN {X 0,Y 533.475,Z 578.191,A -85,B 0,C 180,E1 4623.78,E2 4623.78} C_VEL
LIN {X 0,Y 527.131,Z 563.974,A -85,B 0,C 180,E1 4624.579,E2 4624.579} C_VEL
LIN {X 0,Y 522.102,Z 555.276,A -85,B 0,C 180,E1 4625.769,E2 4625.769} C_VEL
LIN {X 0,Y 520.29,Z 549.53,A -85,B 0,C 180,E1 4626.348,E2 4626.348} C_VEL
LIN {X 0,Y 520.131,Z 549.53,A -85,B 0,C 180,E1 4631.863,E2 4631.863} C_VEL
LIN {X 0,Y 520.205,Z 549.53,A -85,B 0,C 180,E1 4638.154,E2 4638.154} C_VEL
LIN {X 0,Y 520.19,Z 549.53,A -85,B 0,C 180,E1 4644.324,E2 4644.324} C_VEL
LIN {X 0,Y 520.217,Z 549.53,A -85,B 0,C 180,E1 4650.495,E2 4650.495} C_VEL
LIN {X 0,Y 520.383,Z 549.53,A -85,B 0,C 180,E1 4656.957,E2 4656.957} C_VEL
LIN {X 0,Y 520.499,Z 549.762,A -85,B 0,C 180,E1 4657.644,E2 4657.644} C_VEL
LIN {X 0,Y 524.082,Z 570.347,A -85,B 0,C 180,E1 4658.022,E2 4658.022} C_VEL
LIN {X 0,Y 524.062,Z 601.805,A -85,B 0,C 180,E1 4658.689,E2 4658.689} C_VEL
LIN {X 0,Y 523.575,Z 628.589,A -85,B 0,C 180,E1 4659.88,E2 4659.88} C_VEL
LIN {X 0,Y 522.9,Z 654.233,A -85,B 0,C 180,E1 4661.753,E2 4661.753} C_VEL
LIN {X 0,Y 522.219,Z 675.181,A -85,B 0,C 180,E1 4664.071,E2 4664.071} C_VEL
LIN {X 0,Y 521.718,Z 691.716,A -85,B 0,C 180,E1 4666.838,E2 4666.838} C_VEL
LIN {X 0,Y 521.367,Z 703.344,A -85,B 0,C 180,E1 4670.003,E2 4670.003} C_VEL
LIN {X 0,Y 521.214,Z 709.083,A -85,B 0,C 180,E1 4673.354,E2 4673.354} C_VEL
LIN {X 0,Y 521.256,Z 708.866,A -85,B 0,C 180,E1 4676.685,E2 4676.685} C_VEL
LIN {X 0,Y 521.341,Z 702.827,A -85,B 0,C 180,E1 4680.004,E2 4680.004} C_VEL
LIN {X 0,Y 521.634,Z 692.233,A -85,B 0,C 180,E1 4682.877,E2 4682.877} C_VEL
LIN {X 0,Y 522.073,Z 676.322,A -85,B 0,C 180,E1 4685.602,E2 4685.602} C_VEL
LIN {X 0,Y 522.745,Z 655.542,A -85,B 0,C 180,E1 4687.989,E2 4687.989} C_VEL
LIN {X 0,Y 523.452,Z 631.162,A -85,B 0,C 180,E1 4689.86,E2 4689.86} C_VEL
LIN {X 0,Y 524.095,Z 602.663,A -85,B 0,C 180,E1 4691.221,E2 4691.221} C_VEL
LIN {X 0,Y 524.395,Z 573.976,A -85,B 0,C 180,E1 4691.904,E2 4691.904} C_VEL
LIN {X 0,Y 522.627,Z 558.049,A -85,B 0,C 180,E1 4692.182,E2 4692.182} C_VEL
LIN {X 0,Y 520.774,Z 549.53,A -85,B 0,C 180,E1 4692.424,E2 4692.424} C_VEL
LIN {X 0,Y 520.526,Z 549.53,A -85,B 0,C 180,E1 4698.6,E2 4698.6} C_VEL
LIN {X 0,Y 520.361,Z 549.53,A -85,B 0,C 180,E1 4703.958,E2 4703.958} C_VEL
LIN {X 0,Y 520.238,Z 549.53,A -85,B 0,C 180,E1 4709.55,E2 4709.55} C_VEL
LIN {X 0,Y 520.097,Z 549.53,A -85,B 0,C 180,E1 4715.661,E2 4715.661} C_VEL
LIN {X 0,Y 520.105,Z 549.53,A -85,B 0,C 180,E1 4721.866,E2 4721.866} C_VEL
LIN {X 0,Y 520.196,Z 549.53,A -85,B 0,C 180,E1 4728.144,E2 4728.144} C_VEL
LIN {X 0,Y 520.188,Z 549.53,A -85,B 0,C 180,E1 4732.465,E2 4732.465} C_VEL
LIN {X 0,Y 520.165,Z 549.53,A -85,B 0,C 180,E1 4738.518,E2 4738.518} C_VEL
LIN {X 0,Y 520.464,Z 550.2,A -85,B 0,C 180,E1 4743.441,E2 4743.441} C_VEL
LIN {X 0,Y 530.407,Z 577.659,A -85,B 0,C 180,E1 4744.624,E2 4744.624} C_VEL
LIN {X 0,Y 528.984,Z 613.538,A -85,B 0,C 180,E1 4745.913,E2 4745.913} C_VEL
LIN {X 0,Y 527.248,Z 648.135,A -85,B 0,C 180,E1 4747.823,E2 4747.823} C_VEL
LIN {X 0,Y 525.261,Z 680.617,A -85,B 0,C 180,E1 4750.379,E2 4750.379} C_VEL
LIN {X 0,Y 523.657,Z 707.777,A -85,B 0,C 180,E1 4753.25,E2 4753.25} C_VEL
LIN {X 0,Y 522.213,Z 733.026,A -85,B 0,C 180,E1 4756.845,E2 4756.845} C_VEL
LIN {X 0,Y 521.506,Z 751.35,A -85,B 0,C 180,E1 4760.422,E2 4760.422} C_VEL
LIN {X 0,Y 521.086,Z 764.94,A -85,B 0,C 180,E1 4764.182,E2 4764.182} C_VEL
LIN {X 0,Y 521.041,Z 772.682,A -85,B 0,C 180,E1 4767.505,E2 4767.505} C_VEL
LIN {X 0,Y 520.911,Z 777.177,A -85,B 0,C 180,E1 4771.661,E2 4771.661} C_VEL
LIN {X 0,Y 520.961,Z 776.776,A -85,B 0,C 180,E1 4774.986,E2 4774.986} C_VEL
LIN {X 0,Y 521.03,Z 771.273,A -85,B 0,C 180,E1 4779.167,E2 4779.167} C_VEL
LIN {X 0,Y 521.252,Z 759.581,A -85,B 0,C 180,E1 4783.393,E2 4783.393} C_VEL
LIN {X 0,Y 521.853,Z 743.784,A -85,B 0,C 180,E1 4787.106,E2 4787.106} C_VEL
LIN {X 0,Y 522.956,Z 720.945,A -85,B 0,C 180,E1 4790.924,E2 4790.924} C_VEL
LIN {X 0,Y 524.431,Z 694.933,A -85,B 0,C 180,E1 4794.113,E2 4794.113} C_VEL
LIN {X 0,Y 526.215,Z 665.193,A -85,B 0,C 180,E1 4796.854,E2 4796.854} C_VEL
LIN {X 0,Y 528.186,Z 629.25,A -85,B 0,C 180,E1 4799.223,E2 4799.223} C_VEL
LIN {X 0,Y 529.728,Z 593.016,A -85,B 0,C 180,E1 4800.819,E2 4800.819} C_VEL
LIN {X 0,Y 529.758,Z 574.818,A -85,B 0,C 180,E1 4801.406,E2 4801.406} C_VEL
LIN {X 0,Y 520.468,Z 549.53,A -85,B 0,C 180,E1 4802.523,E2 4802.523} C_VEL
LIN {X 0,Y 520.25,Z 549.53,A -85,B 0,C 180,E1 4808.443,E2 4808.443} C_VEL
LIN {X 0,Y 520.08,Z 549.53,A -85,B 0,C 180,E1 4814.142,E2 4814.142} C_VEL
LIN {X 0,Y 520.243,Z 549.53,A -85,B 0,C 180,E1 4820.342,E2 4820.342} C_VEL
LIN {X 0,Y 520.422,Z 549.53,A -85,B 0,C 180,E1 4826.565,E2 4826.565} C_VEL
LIN {X 0,Y 520.216,Z 549.53,A -85,B 0,C 180,E1 4832.342,E2 4832.342} C_VEL
LIN {X 0,Y 520.296,Z 549.53,A -85,B 0,C 180,E1 4838.156,E2 4838.156} C_VEL
LIN {X 0,Y 520.418,Z 549.53,A -85,B 0,C 180,E1 4840.986,E2 4840.986} C_VEL
LIN {X 0,Y 523.572,Z 577.412,A -85,B 0,C 180,E1 4841.478,E2 4841.478} C_VEL
LIN {X 0,Y 523.391,Z 615.893,A -85,B 0,C 180,E1 4842.167,E2 4842.167} C_VEL
LIN {X 0,Y 523.02,Z 640.5,A -85,B 0,C 180,E1 4843.227,E2 4843.227} C_VEL
LIN {X 0,Y 522.45,Z 663.863,A -85,B 0,C 180,E1 4844.929,E2 4844.929} C_VEL
LIN {X 0,Y 521.935,Z 682.585,A -85,B 0,C 180,E1 4847.048,E2 4847.048} C_VEL
LIN {X 0,Y 521.598,Z 697.41,A -85,B 0,C 180,E1 4849.658,E2 4849.658} C_VEL
LIN {X 0,Y 521.381,Z 706.795,A -85,B 0,C 180,E1 4852.519,E2 4852.519} C_VEL
LIN {X 0,Y 521.311,Z 710.337,A -85,B 0,C 180,E1 4855.014,E2 4855.014} C_VEL
LIN {X 0,Y 521.315,Z 710.517,A -85,B 0,C 180,E1 4856.677,E2 4856.677} C_VEL
LIN {X 0,Y 521.439,Z 707.486,A -85,B 0,C 180,E1 4859.167,E2 4859.167} C_VEL
LIN {X 0,Y 521.649,Z 698.59,A -85,B 0,C 180,E1 4862.068,E2 4862.068} C_VEL
LIN {X 0,Y 522.004,Z 684.749,A -85,B 0,C 180,E1 4864.623,E2 4864.623} C_VEL
LIN {X 0,Y 522.527,Z 665.932,A -85,B 0,C 180,E1 4866.838,E2 4866.838} C_VEL
LIN {X 0,Y 523.01,Z 644.128,A -85,B 0,C 180,E1 4868.5,E2 4868.5} C_VEL
LIN {X 0,Y 523.43,Z 619.077,A -85,B 0,C 180,E1 4869.643,E2 4869.643} C_VEL
LIN {X 0,Y 523.5,Z 586.101,A -85,B 0,C 180,E1 4870.287,E2 4870.287} C_VEL
LIN {X 0,Y 522.532,Z 557.873,A -85,B 0,C 180,E1 4870.707,E2 4870.707} C_VEL
LIN {X 0,Y 520.769,Z 549.53,A -85,B 0,C 180,E1 4870.987,E2 4870.987} C_VEL
LIN {X 0,Y 520.462,Z 549.53,A -85,B 0,C 180,E1 4876.882,E2 4876.882} C_VEL
LIN {X 0,Y 520.331,Z 549.53,A -85,B 0,C 180,E1 4882.145,E2 4882.145} C_VEL
LIN {X 0,Y 520.273,Z 549.53,A -85,B 0,C 180,E1 4884.012,E2 4884.012} C_VEL
LIN {X 0,Y 516.144,Z 549.53,A -85,B 0,C 180,E1 4885.895,E2 4885.895} C_VEL
LIN {X 0,Y 512.272,Z 549.53,A -85,B 0,C 180,E1 4887.808,E2 4887.808} C_VEL
LIN {X 0,Y 512.166,Z 549.53,A -85,B 0,C 180,E1 4894.038,E2 4894.038} C_VEL
LIN {X 0,Y 512.316,Z 549.53,A -85,B 0,C 180,E1 4900.012,E2 4900.012} C_VEL
LIN {X 0,Y 512.234,Z 549.53,A -85,B 0,C 180,E1 4905,E2 4905} C_VEL
LIN {X 0,Y 512.183,Z 549.53,A -85,B 0,C 180,E1 4911.773,E2 4911.773} C_VEL
LIN {X 0,Y 512.259,Z 549.689,A -85,B 0,C 180,E1 4913.066,E2 4913.066} C_VEL
LIN {X 0,Y 517.421,Z 563.797,A -85,B 0,C 180,E1 4914.364,E2 4914.364} C_VEL
LIN {X 0,Y 522.572,Z 571.41,A -85,B 0,C 180,E1 4915.305,E2 4915.305} C_VEL
LIN {X 0,Y 527.539,Z 582.274,A -85,B 0,C 180,E1 4915.853,E2 4915.853} C_VEL
LIN {X 0,Y 526.681,Z 628.211,A -85,B 0,C 180,E1 4916.751,E2 4916.751} C_VEL
LIN {X 0,Y 524.956,Z 665.746,A -85,B 0,C 180,E1 4918.107,E2 4918.107} C_VEL
LIN {X 0,Y 522.584,Z 702.756,A -85,B 0,C 180,E1 4920.115,E2 4920.115} C_VEL
LIN {X 0,Y 519.948,Z 738.182,A -85,B 0,C 180,E1 4922.796,E2 4922.796} C_VEL
LIN {X 0,Y 517.571,Z 768.978,A -85,B 0,C 180,E1 4925.906,E2 4925.906} C_VEL
LIN {X 0,Y 515.538,Z 796.96,A -85,B 0,C 180,E1 4929.623,E2 4929.623} C_VEL
LIN {X 0,Y 514.103,Z 819.458,A -85,B 0,C 180,E1 4933.587,E2 4933.587} C_VEL
LIN {X 0,Y 513.392,Z 836.552,A -85,B 0,C 180,E1 4937.694,E2 4937.694} C_VEL
LIN {X 0,Y 513.154,Z 847.714,A -85,B 0,C 180,E1 4941.544,E2 4941.544} C_VEL
LIN {X 0,Y 512.999,Z 853.987,A -85,B 0,C 180,E1 4944.936,E2 4944.936} C_VEL
LIN {X 0,Y 512.99,Z 857.11,A -85,B 0,C 180,E1 4948.314,E2 4948.314} C_VEL
LIN {X 0,Y 513.101,Z 857.11,A -85,B 0,C 180,E1 4951.685,E2 4951.685} C_VEL
LIN {X 0,Y 513.099,Z 852.744,A -85,B 0,C 180,E1 4955.909,E2 4955.909} C_VEL
LIN {X 0,Y 513.197,Z 843.328,A -85,B 0,C 180,E1 4960.162,E2 4960.162} C_VEL
LIN {X 0,Y 513.733,Z 829.186,A -85,B 0,C 180,E1 4964.241,E2 4964.241} C_VEL
LIN {X 0,Y 514.809,Z 809.37,A -85,B 0,C 180,E1 4968.329,E2 4968.329} C_VEL
LIN {X 0,Y 516.523,Z 783.298,A -85,B 0,C 180,E1 4972.323,E2 4972.323} C_VEL
LIN {X 0,Y 518.842,Z 752.45,A -85,B 0,C 180,E1 4975.868,E2 4975.868} C_VEL
LIN {X 0,Y 521.367,Z 718.916,A -85,B 0,C 180,E1 4978.766,E2 4978.766} C_VEL
LIN {X 0,Y 523.981,Z 681.616,A -85,B 0,C 180,E1 4981.12,E2 4981.12} C_VEL
LIN {X 0,Y 526.029,Z 644.293,A -85,B 0,C 180,E1 4982.743,E2 4982.743} C_VEL
LIN {X 0,Y 527.469,Z 606.036,A -85,B 0,C 180,E1 4983.749,E2 4983.749} C_VEL
LIN {X 0,Y 526.902,Z 580.711,A -85,B 0,C 180,E1 4984.219,E2 4984.219} C_VEL
LIN {X 0,Y 521.156,Z 567.776,A -85,B 0,C 180,E1 4984.968,E2 4984.968} C_VEL
LIN {X 0,Y 515.145,Z 558.56,A -85,B 0,C 180,E1 4985.968,E2 4985.968} C_VEL
LIN {X 0,Y 512.378,Z 549.53,A -85,B 0,C 180,E1 4986.781,E2 4986.781} C_VEL
LIN {X 0,Y 512.186,Z 549.53,A -85,B 0,C 180,E1 4992.664,E2 4992.664} C_VEL
LIN {X 0,Y 512.268,Z 549.53,A -85,B 0,C 180,E1 4997.435,E2 4997.435} C_VEL
LIN {X 0,Y 512.303,Z 549.53,A -85,B 0,C 180,E1 5002.691,E2 5002.691} C_VEL
LIN {X 0,Y 512.297,Z 549.53,A -85,B 0,C 180,E1 5008.683,E2 5008.683} C_VEL
LIN {X 0,Y 512.354,Z 549.53,A -85,B 0,C 180,E1 5013.786,E2 5013.786} C_VEL
LIN {X 0,Y 512.539,Z 549.53,A -85,B 0,C 180,E1 5017.4,E2 5017.4} C_VEL
LIN {X 0,Y 516.427,Z 571.541,A -85,B 0,C 180,E1 5017.837,E2 5017.837} C_VEL
LIN {X 0,Y 516.401,Z 603.999,A -85,B 0,C 180,E1 5018.537,E2 5018.537} C_VEL
LIN {X 0,Y 515.871,Z 631.274,A -85,B 0,C 180,E1 5019.789,E2 5019.789} C_VEL
LIN {X 0,Y 515.229,Z 655.94,A -85,B 0,C 180,E1 5021.631,E2 5021.631} C_VEL
LIN {X 0,Y 514.579,Z 675.71,A -85,B 0,C 180,E1 5023.828,E2 5023.828} C_VEL
LIN {X 0,Y 514.008,Z 692.613,A -85,B 0,C 180,E1 5026.637,E2 5026.637} C_VEL
LIN {X 0,Y 513.629,Z 704.5,A -85,B 0,C 180,E1 5029.851,E2 5029.851} C_VEL
LIN {X 0,Y 513.449,Z 710.367,A -85,B 0,C 180,E1 5033.253,E2 5033.253} C_VEL
LIN {X 0,Y 513.488,Z 710.248,A -85,B 0,C 180,E1 5036.634,E2 5036.634} C_VEL
LIN {X 0,Y 513.584,Z 704.24,A -85,B 0,C 180,E1 5040.004,E2 5040.004} C_VEL
LIN {X 0,Y 513.91,Z 692.431,A -85,B 0,C 180,E1 5043.181,E2 5043.181} C_VEL
LIN {X 0,Y 514.406,Z 676.304,A -85,B 0,C 180,E1 5045.897,E2 5045.897} C_VEL
LIN {X 0,Y 515.186,Z 654.783,A -85,B 0,C 180,E1 5048.319,E2 5048.319} C_VEL
LIN {X 0,Y 515.89,Z 629.571,A -85,B 0,C 180,E1 5050.205,E2 5050.205} C_VEL
LIN {X 0,Y 516.474,Z 601.551,A -85,B 0,C 180,E1 5051.495,E2 5051.495} C_VEL
LIN {X 0,Y 516.688,Z 569.665,A -85,B 0,C 180,E1 5052.191,E2 5052.191} C_VEL
LIN {X 0,Y 512.888,Z 549.53,A -85,B 0,C 180,E1 5052.608,E2 5052.608} C_VEL
LIN {X 0,Y 512.582,Z 549.53,A -85,B 0,C 180,E1 5058.899,E2 5058.899} C_VEL
LIN {X 0,Y 512.41,Z 549.53,A -85,B 0,C 180,E1 5064.353,E2 5064.353} C_VEL
LIN {X 0,Y 512.274,Z 549.53,A -85,B 0,C 180,E1 5070.056,E2 5070.056} C_VEL
LIN {X 0,Y 512.138,Z 549.53,A -85,B 0,C 180,E1 5076.112,E2 5076.112} C_VEL
LIN {X 0,Y 512.164,Z 549.53,A -85,B 0,C 180,E1 5082.552,E2 5082.552} C_VEL
LIN {X 0,Y 512.253,Z 549.53,A -85,B 0,C 180,E1 5087.437,E2 5087.437} C_VEL
LIN {X 0,Y 512.252,Z 549.53,A -85,B 0,C 180,E1 5092.698,E2 5092.698} C_VEL
LIN {X 0,Y 512.246,Z 549.53,A -85,B 0,C 180,E1 5098.691,E2 5098.691} C_VEL
LIN {X 0,Y 512.461,Z 549.53,A -85,B 0,C 180,E1 5102.911,E2 5102.911} C_VEL
LIN {X 0,Y 523.396,Z 579.275,A -85,B 0,C 180,E1 5104.26,E2 5104.26} C_VEL
LIN {X 0,Y 521.847,Z 614.589,A -85,B 0,C 180,E1 5105.562,E2 5105.562} C_VEL
LIN {X 0,Y 519.975,Z 648.847,A -85,B 0,C 180,E1 5107.496,E2 5107.496} C_VEL
LIN {X 0,Y 517.742,Z 682.299,A -85,B 0,C 180,E1 5110.193,E2 5110.193} C_VEL
LIN {X 0,Y 515.913,Z 709.815,A -85,B 0,C 180,E1 5113.21,E2 5113.21} C_VEL
LIN {X 0,Y 514.401,Z 734.583,A -85,B 0,C 180,E1 5116.858,E2 5116.858} C_VEL
LIN {X 0,Y 513.607,Z 753.308,A -85,B 0,C 180,E1 5120.7,E2 5120.7} C_VEL
LIN {X 0,Y 513.197,Z 766.265,A -85,B 0,C 180,E1 5124.516,E2 5124.516} C_VEL
LIN {X 0,Y 513.06,Z 774.072,A -85,B 0,C 180,E1 5128.315,E2 5128.315} C_VEL
LIN {X 0,Y 513.009,Z 777.188,A -85,B 0,C 180,E1 5131.686,E2 5131.686} C_VEL
LIN {X 0,Y 513.052,Z 776.741,A -85,B 0,C 180,E1 5135.063,E2 5135.063} C_VEL
LIN {X 0,Y 513.155,Z 771.324,A -85,B 0,C 180,E1 5139.235,E2 5139.235} C_VEL
LIN {X 0,Y 513.349,Z 760.867,A -85,B 0,C 180,E1 5143.17,E2 5143.17} C_VEL
LIN {X 0,Y 514.035,Z 745.051,A -85,B 0,C 180,E1 5147.074,E2 5147.074} C_VEL
LIN {X 0,Y 515.179,Z 723.558,A -85,B 0,C 180,E1 5150.806,E2 5150.806} C_VEL
LIN {X 0,Y 516.72,Z 697.719,A -85,B 0,C 180,E1 5154.136,E2 5154.136} C_VEL
LIN {X 0,Y 518.819,Z 666.004,A -85,B 0,C 180,E1 5157.149,E2 5157.149} C_VEL
LIN {X 0,Y 520.901,Z 631.086,A -85,B 0,C 180,E1 5159.507,E2 5159.507} C_VEL
LIN {X 0,Y 522.627,Z 595.682,A -85,B 0,C 180,E1 5161.132,E2 5161.132} C_VEL
LIN {X 0,Y 522.696,Z 576.965,A -85,B 0,C 180,E1 5161.756,E2 5161.756} C_VEL
LIN {X 0,Y 512.528,Z 549.53,A -85,B 0,C 180,E1 5163.017,E2 5163.017} C_VEL
LIN {X 0,Y 512.346,Z 549.53,A -85,B 0,C 180,E1 5168.213,E2 5168.213} C_VEL
LIN {X 0,Y 512.144,Z 549.53,A -85,B 0,C 180,E1 5174.99,E2 5174.99} C_VEL
LIN {X 0,Y 512.32,Z 549.53,A -85,B 0,C 180,E1 5179.988,E2 5179.988} C_VEL
LIN {X 0,Y 512.437,Z 549.53,A -85,B 0,C 180,E1 5185.973,E2 5185.973} C_VEL
LIN {X 0,Y 512.292,Z 549.53,A -85,B 0,C 180,E1 5192.102,E2 5192.102} C_VEL
LIN {X 0,Y 512.293,Z 549.53,A -85,B 0,C 180,E1 5197.48,E2 5197.48} C_VEL
LIN {X 0,Y 512.487,Z 549.53,A -85,B 0,C 180,E1 5200.762,E2 5200.762} C_VEL
LIN {X 0,Y 515.895,Z 574.172,A -85,B 0,C 180,E1 5201.227,E2 5201.227} C_VEL
LIN {X 0,Y 515.751,Z 615.398,A -85,B 0,C 180,E1 5201.941,E2 5201.941} C_VEL
LIN {X 0,Y 515.373,Z 640.001,A -85,B 0,C 180,E1 5202.97,E2 5202.97} C_VEL
LIN {X 0,Y 514.807,Z 664.042,A -85,B 0,C 180,E1 5204.7,E2 5204.7} C_VEL
LIN {X 0,Y 514.216,Z 683.154,A -85,B 0,C 180,E1 5206.85,E2 5206.85} C_VEL
LIN {X 0,Y 513.865,Z 698.28,A -85,B 0,C 180,E1 5209.5,E2 5209.5} C_VEL
LIN {X 0,Y 513.6,Z 707.882,A -85,B 0,C 180,E1 5212.398,E2 5212.398} C_VEL
LIN {X 0,Y 513.517,Z 711.589,A -85,B 0,C 180,E1 5214.938,E2 5214.938} C_VEL
LIN {X 0,Y 513.515,Z 711.045,A -85,B 0,C 180,E1 5217.762,E2 5217.762} C_VEL
LIN {X 0,Y 513.742,Z 704.669,A -85,B 0,C 180,E1 5220.838,E2 5220.838} C_VEL
LIN {X 0,Y 514.054,Z 693.789,A -85,B 0,C 180,E1 5223.447,E2 5223.447} C_VEL
LIN {X 0,Y 514.583,Z 677.431,A -85,B 0,C 180,E1 5225.887,E2 5225.887} C_VEL
LIN {X 0,Y 515.111,Z 656.665,A -85,B 0,C 180,E1 5227.889,E2 5227.889} C_VEL
LIN {X 0,Y 515.586,Z 631.942,A -85,B 0,C 180,E1 5229.366,E2 5229.366} C_VEL
LIN {X 0,Y 515.788,Z 604.767,A -85,B 0,C 180,E1 5230.207,E2 5230.207} C_VEL
LIN {X 0,Y 514.927,Z 559.198,A -85,B 0,C 180,E1 5230.889,E2 5230.889} C_VEL
LIN {X 0,Y 512.843,Z 549.53,A -85,B 0,C 180,E1 5231.17,E2 5231.17} C_VEL
LIN {X 0,Y 512.557,Z 549.53,A -85,B 0,C 180,E1 5237.118,E2 5237.118} C_VEL
LIN {X 0,Y 512.38,Z 549.53,A -85,B 0,C 180,E1 5242.507,E2 5242.507} C_VEL
LIN {X 0,Y 512.272,Z 549.53,A -85,B 0,C 180,E1 5247.808,E2 5247.808} C_VEL
LIN {X 0,Y 509.768,Z 549.53,A -85,B 0,C 180,E1 5249.252,E2 5249.252} C_VEL
LIN {X 0,Y 504.276,Z 549.53,A -85,B 0,C 180,E1 5251.416,E2 5251.416} C_VEL
LIN {X 0,Y 504.178,Z 549.53,A -85,B 0,C 180,E1 5251.666,E2 5251.666} C_VEL
LIN {X 0,Y 504.313,Z 549.53,A -85,B 0,C 180,E1 5256.754,E2 5256.754} C_VEL
LIN {X 0,Y 504.295,Z 549.53,A -85,B 0,C 180,E1 5261.568,E2 5261.568} C_VEL
LIN {X 0,Y 504.198,Z 549.53,A -85,B 0,C 180,E1 5266.493,E2 5266.493} C_VEL
LIN {X 0,Y 504.326,Z 549.806,A -85,B 0,C 180,E1 5272.641,E2 5272.641} C_VEL
LIN {X 0,Y 509.821,Z 566.658,A -85,B 0,C 180,E1 5274.184,E2 5274.184} C_VEL
LIN {X 0,Y 517.668,Z 577.428,A -85,B 0,C 180,E1 5275.03,E2 5275.03} C_VEL
LIN {X 0,Y 520.898,Z 584.17,A -85,B 0,C 180,E1 5275.388,E2 5275.388} C_VEL
LIN {X 0,Y 520.01,Z 629.6,A -85,B 0,C 180,E1 5276.312,E2 5276.312} C_VEL
LIN {X 0,Y 518.119,Z 667.036,A -85,B 0,C 180,E1 5277.697,E2 5277.697} C_VEL
LIN {X 0,Y 515.494,Z 704.485,A -85,B 0,C 180,E1 5279.782,E2 5279.782} C_VEL
LIN {X 0,Y 512.643,Z 739.459,A -85,B 0,C 180,E1 5282.495,E2 5282.495} C_VEL
LIN {X 0,Y 509.915,Z 771.719,A -85,B 0,C 180,E1 5285.858,E2 5285.858} C_VEL
LIN {X 0,Y 507.712,Z 799.513,A -85,B 0,C 180,E1 5289.701,E2 5289.701} C_VEL
LIN {X 0,Y 506.245,Z 821.561,A -85,B 0,C 180,E1 5293.77,E2 5293.77} C_VEL
LIN {X 0,Y 505.495,Z 838.03,A -85,B 0,C 180,E1 5297.937,E2 5297.937} C_VEL
LIN {X 0,Y 505.213,Z 849.598,A -85,B 0,C 180,E1 5302.274,E2 5302.274} C_VEL
LIN {X 0,Y 505.081,Z 855.944,A -85,B 0,C 180,E1 5306.574,E2 5306.574} C_VEL
LIN {X 0,Y 505.099,Z 857.5,A -85,B 0,C 180,E1 5310,E2 5310} C_VEL
LIN {X 0,Y 505.085,Z 855.944,A -85,B 0,C 180,E1 5313.426,E2 5313.426} C_VEL
LIN {X 0,Y 505.227,Z 849.6,A -85,B 0,C 180,E1 5317.725,E2 5317.725} C_VEL
LIN {X 0,Y 505.577,Z 838.032,A -85,B 0,C 180,E1 5322.061,E2 5322.061} C_VEL
LIN {X 0,Y 506.471,Z 820.516,A -85,B 0,C 180,E1 5326.444,E2 5326.444} C_VEL
LIN {X 0,Y 507.973,Z 796.856,A -85,B 0,C 180,E1 5330.71,E2 5330.71} C_VEL
LIN {X 0,Y 510.206,Z 768.988,A -85,B 0,C 180,E1 5334.463,E2 5334.463} C_VEL
LIN {X 0,Y 512.882,Z 736.553,A -85,B 0,C 180,E1 5337.761,E2 5337.761} C_VEL
LIN {X 0,Y 515.76,Z 700.891,A -85,B 0,C 180,E1 5340.45,E2 5340.45} C_VEL
LIN {X 0,Y 518.286,Z 663.189,A -85,B 0,C 180,E1 5342.476,E2 5342.476} C_VEL
LIN {X 0,Y 520.171,Z 625.166,A -85,B 0,C 180,E1 5343.809,E2 5343.809} C_VEL
LIN {X 0,Y 520.524,Z 583.769,A -85,B 0,C 180,E1 5344.647,E2 5344.647} C_VEL
LIN {X 0,Y 513.219,Z 570.763,A -85,B 0,C 180,E1 5345.393,E2 5345.393} C_VEL
LIN {X 0,Y 506.642,Z 558.201,A -85,B 0,C 180,E1 5346.474,E2 5346.474} C_VEL
LIN {X 0,Y 504.477,Z 549.53,A -85,B 0,C 180,E1 5347.261,E2 5347.261} C_VEL
LIN {X 0,Y 504.24,Z 549.53,A -85,B 0,C 180,E1 5354.096,E2 5354.096} C_VEL
LIN {X 0,Y 504.305,Z 549.53,A -85,B 0,C 180,E1 5358.834,E2 5358.834} C_VEL
LIN {X 0,Y 504.398,Z 549.53,A -85,B 0,C 180,E1 5363.886,E2 5363.886} C_VEL
LIN {X 0,Y 504.344,Z 549.53,A -85,B 0,C 180,E1 5370.202,E2 5370.202} C_VEL
LIN {X 0,Y 504.43,Z 549.53,A -85,B 0,C 180,E1 5375.244,E2 5375.244} C_VEL
LIN {X 0,Y 504.628,Z 549.53,A -85,B 0,C 180,E1 5377.179,E2 5377.179} C_VEL
LIN {X 0,Y 508.752,Z 572.01,A -85,B 0,C 180,E1 5377.634,E2 5377.634} C_VEL
LIN {X 0,Y 508.756,Z 604.182,A -85,B 0,C 180,E1 5378.315,E2 5378.315} C_VEL
LIN {X 0,Y 508.275,Z 631.208,A -85,B 0,C 180,E1 5379.529,E2 5379.529} C_VEL
LIN {X 0,Y 507.675,Z 655.202,A -85,B 0,C 180,E1 5381.284,E2 5381.284} C_VEL
LIN {X 0,Y 506.91,Z 676.191,A -85,B 0,C 180,E1 5383.576,E2 5383.576} C_VEL
LIN {X 0,Y 506.336,Z 692.448,A -85,B 0,C 180,E1 5386.211,E2 5386.211} C_VEL
LIN {X 0,Y 505.957,Z 704.386,A -85,B 0,C 180,E1 5389.261,E2 5389.261} C_VEL
LIN {X 0,Y 505.667,Z 710.742,A -85,B 0,C 180,E1 5392.286,E2 5392.286} C_VEL
LIN {X 0,Y 505.666,Z 712.396,A -85,B 0,C 180,E1 5394.868,E2 5394.868} C_VEL
LIN {X 0,Y 505.704,Z 709.409,A -85,B 0,C 180,E1 5398.294,E2 5398.294} C_VEL
LIN {X 0,Y 505.943,Z 701.959,A -85,B 0,C 180,E1 5401.225,E2 5401.225} C_VEL
LIN {X 0,Y 506.305,Z 688.576,A -85,B 0,C 180,E1 5404.277,E2 5404.277} C_VEL
LIN {X 0,Y 506.993,Z 669.485,A -85,B 0,C 180,E1 5407.056,E2 5407.056} C_VEL
LIN {X 0,Y 507.835,Z 646.413,A -85,B 0,C 180,E1 5409.302,E2 5409.302} C_VEL
LIN {X 0,Y 508.518,Z 619.595,A -85,B 0,C 180,E1 5410.996,E2 5410.996} C_VEL
LIN {X 0,Y 509.086,Z 590.871,A -85,B 0,C 180,E1 5412.043,E2 5412.043} C_VEL
LIN {X 0,Y 508.271,Z 564.286,A -85,B 0,C 180,E1 5412.528,E2 5412.528} C_VEL
LIN {X 0,Y 504.914,Z 549.53,A -85,B 0,C 180,E1 5412.917,E2 5412.917} C_VEL
LIN {X 0,Y 504.656,Z 549.53,A -85,B 0,C 180,E1 5419.208,E2 5419.208} C_VEL
LIN {X 0,Y 504.45,Z 549.53,A -85,B 0,C 180,E1 5424.763,E2 5424.763} C_VEL
LIN {X 0,Y 504.362,Z 549.53,A -85,B 0,C 180,E1 5430.577,E2 5430.577} C_VEL
LIN {X 0,Y 504.212,Z 549.53,A -85,B 0,C 180,E1 5436.772,E2 5436.772} C_VEL
LIN {X 0,Y 504.187,Z 549.53,A -85,B 0,C 180,E1 5443.508,E2 5443.508} C_VEL
LIN {X 0,Y 504.298,Z 549.53,A -85,B 0,C 180,E1 5448.824,E2 5448.824} C_VEL
LIN {X 0,Y 504.319,Z 549.53,A -85,B 0,C 180,E1 5453.898,E2 5453.898} C_VEL
LIN {X 0,Y 504.332,Z 549.53,A -85,B 0,C 180,E1 5460.203,E2 5460.203} C_VEL
LIN {X 0,Y 504.486,Z 549.53,A -85,B 0,C 180,E1 5462.426,E2 5462.426} C_VEL
LIN {X 0,Y 516.379,Z 580.533,A -85,B 0,C 180,E1 5463.883,E2 5463.883} C_VEL
LIN {X 0,Y 514.788,Z 615.372,A -85,B 0,C 180,E1 5465.187,E2 5465.187} C_VEL
LIN {X 0,Y 512.711,Z 649.682,A -85,B 0,C 180,E1 5467.159,E2 5467.159} C_VEL
LIN {X 0,Y 510.201,Z 683.983,A -85,B 0,C 180,E1 5470,E2 5470} C_VEL
LIN {X 0,Y 508.171,Z 711.839,A -85,B 0,C 180,E1 5473.169,E2 5473.169} C_VEL
LIN {X 0,Y 506.65,Z 734.848,A -85,B 0,C 180,E1 5476.653,E2 5476.653} C_VEL
LIN {X 0,Y 505.752,Z 753.827,A -85,B 0,C 180,E1 5480.635,E2 5480.635} C_VEL
LIN {X 0,Y 505.305,Z 766.392,A -85,B 0,C 180,E1 5484.43,E2 5484.43} C_VEL
LIN {X 0,Y 505.163,Z 774.132,A -85,B 0,C 180,E1 5488.288,E2 5488.288} C_VEL
LIN {X 0,Y 505.107,Z 777.199,A -85,B 0,C 180,E1 5491.712,E2 5491.712} C_VEL
LIN {X 0,Y 505.143,Z 776.706,A -85,B 0,C 180,E1 5495.143,E2 5495.143} C_VEL
LIN {X 0,Y 505.258,Z 771.654,A -85,B 0,C 180,E1 5499.152,E2 5499.152} C_VEL
LIN {X 0,Y 505.483,Z 760.703,A -85,B 0,C 180,E1 5503.379,E2 5503.379} C_VEL
LIN {X 0,Y 506.236,Z 744.265,A -85,B 0,C 180,E1 5507.456,E2 5507.456} C_VEL
LIN {X 0,Y 507.571,Z 721.768,A -85,B 0,C 180,E1 5511.361,E2 5511.361} C_VEL
LIN {X 0,Y 509.314,Z 696.099,A -85,B 0,C 180,E1 5514.64,E2 5514.64} C_VEL
LIN {X 0,Y 511.56,Z 665.088,A -85,B 0,C 180,E1 5517.596,E2 5517.596} C_VEL
LIN {X 0,Y 513.892,Z 630.51,A -85,B 0,C 180,E1 5519.951,E2 5519.951} C_VEL
LIN {X 0,Y 515.653,Z 594.798,A -85,B 0,C 180,E1 5521.579,E2 5521.579} C_VEL
LIN {X 0,Y 515.532,Z 578.657,A -85,B 0,C 180,E1 5522.135,E2 5522.135} C_VEL
LIN {X 0,Y 504.573,Z 549.53,A -85,B 0,C 180,E1 5523.527,E2 5523.527} C_VEL
LIN {X 0,Y 504.389,Z 549.53,A -85,B 0,C 180,E1 5528.928,E2 5528.928} C_VEL
LIN {X 0,Y 504.158,Z 549.53,A -85,B 0,C 180,E1 5534.075,E2 5534.075} C_VEL
LIN {X 0,Y 504.271,Z 549.53,A -85,B 0,C 180,E1 5538.821,E2 5538.821} C_VEL
LIN {X 0,Y 504.51,Z 549.53,A -85,B 0,C 180,E1 5545.363,E2 5545.363} C_VEL
LIN {X 0,Y 504.356,Z 549.53,A -85,B 0,C 180,E1 5551.394,E2 5551.394} C_VEL
LIN {X 0,Y 504.382,Z 549.53,A -85,B 0,C 180,E1 5557.107,E2 5557.107} C_VEL
LIN {X 0,Y 504.577,Z 549.53,A -85,B 0,C 180,E1 5560.511,E2 5560.511} C_VEL
LIN {X 0,Y 508.224,Z 574.106,A -85,B 0,C 180,E1 5561.016,E2 5561.016} C_VEL
LIN {X 0,Y 508.05,Z 617.062,A -85,B 0,C 180,E1 5561.775,E2 5561.775} C_VEL
LIN {X 0,Y 507.632,Z 643.252,A -85,B 0,C 180,E1 5562.925,E2 5562.925} C_VEL
LIN {X 0,Y 507.031,Z 666.702,A -85,B 0,C 180,E1 5564.695,E2 5564.695} C_VEL
LIN {X 0,Y 506.45,Z 685.28,A -85,B 0,C 180,E1 5566.864,E2 5566.864} C_VEL
LIN {X 0,Y 506.141,Z 698.788,A -85,B 0,C 180,E1 5569.257,E2 5569.257} C_VEL
LIN {X 0,Y 505.82,Z 708.983,A -85,B 0,C 180,E1 5572.281,E2 5572.281} C_VEL
LIN {X 0,Y 505.732,Z 712.839,A -85,B 0,C 180,E1 5574.86,E2 5574.86} C_VEL
LIN {X 0,Y 505.761,Z 713.189,A -85,B 0,C 180,E1 5576.575,E2 5576.575} C_VEL
LIN {X 0,Y 505.91,Z 709.789,A -85,B 0,C 180,E1 5579.421,E2 5579.421} C_VEL
LIN {X 0,Y 506.148,Z 701.675,A -85,B 0,C 180,E1 5582.126,E2 5582.126} C_VEL
LIN {X 0,Y 506.596,Z 687.027,A -85,B 0,C 180,E1 5584.909,E2 5584.909} C_VEL
LIN {X 0,Y 507.202,Z 668.211,A -85,B 0,C 180,E1 5587.153,E2 5587.153} C_VEL
LIN {X 0,Y 507.692,Z 645.954,A -85,B 0,C 180,E1 5588.866,E2 5588.866} C_VEL
LIN {X 0,Y 508.063,Z 621.529,A -85,B 0,C 180,E1 5589.991,E2 5589.991} C_VEL
LIN {X 0,Y 508.121,Z 587.586,A -85,B 0,C 180,E1 5590.662,E2 5590.662} C_VEL
LIN {X 0,Y 507.465,Z 561.25,A -85,B 0,C 180,E1 5591.064,E2 5591.064} C_VEL
LIN {X 0,Y 504.894,Z 549.53,A -85,B 0,C 180,E1 5591.378,E2 5591.378} C_VEL
LIN {X 0,Y 504.625,Z 549.53,A -85,B 0,C 180,E1 5597.396,E2 5597.396} C_VEL
LIN {X 0,Y 504.448,Z 549.53,A -85,B 0,C 180,E1 5602.881,E2 5602.881} C_VEL
LIN {X 0,Y 504.287,Z 549.53,A -85,B 0,C 180,E1 5608.602,E2 5608.602} C_VEL
LIN {X 0,Y 504.178,Z 549.53,A -85,B 0,C 180,E1 5611.666,E2 5611.666} C_VEL
LIN {X 0,Y 500.323,Z 549.53,A -85,B 0,C 180,E1 5613.608,E2 5613.608} C_VEL
LIN {X 0,Y 496.331,Z 549.53,A -85,B 0,C 180,E1 5615.579,E2 5615.579} C_VEL
LIN {X 0,Y 496.348,Z 549.53,A -85,B 0,C 180,E1 5621.974,E2 5621.974} C_VEL
LIN {X 0,Y 496.25,Z 549.53,A -85,B 0,C 180,E1 5628.005,E2 5628.005} C_VEL
LIN {X 0,Y 496.408,Z 550.112,A -85,B 0,C 180,E1 5632.214,E2 5632.214} C_VEL
LIN {X 0,Y 501.614,Z 567.46,A -85,B 0,C 180,E1 5633.706,E2 5633.706} C_VEL
LIN {X 0,Y 512.954,Z 584.085,A -85,B 0,C 180,E1 5634.807,E2 5634.807} C_VEL
LIN {X 0,Y 514.389,Z 587.421,A -85,B 0,C 180,E1 5634.961,E2 5634.961} C_VEL
LIN {X 0,Y 513.389,Z 630.416,A -85,B 0,C 180,E1 5635.846,E2 5635.846} C_VEL
LIN {X 0,Y 511.235,Z 669.271,A -85,B 0,C 180,E1 5637.324,E2 5637.324} C_VEL
LIN {X 0,Y 508.393,Z 706.427,A -85,B 0,C 180,E1 5639.455,E2 5639.455} C_VEL
LIN {X 0,Y 505.242,Z 741.938,A -85,B 0,C 180,E1 5642.297,E2 5642.297} C_VEL
LIN {X 0,Y 502.345,Z 773.717,A -85,B 0,C 180,E1 5645.722,E2 5645.722} C_VEL
LIN {X 0,Y 500.003,Z 800.795,A -85,B 0,C 180,E1 5649.592,E2 5649.592} C_VEL
LIN {X 0,Y 498.412,Z 822.551,A -85,B 0,C 180,E1 5653.734,E2 5653.734} C_VEL
LIN {X 0,Y 497.64,Z 838.029,A -85,B 0,C 180,E1 5657.743,E2 5657.743} C_VEL
LIN {X 0,Y 497.328,Z 849.598,A -85,B 0,C 180,E1 5662.151,E2 5662.151} C_VEL
LIN {X 0,Y 497.19,Z 855.945,A -85,B 0,C 180,E1 5666.519,E2 5666.519} C_VEL
LIN {X 0,Y 497.226,Z 857.5,A -85,B 0,C 180,E1 5670,E2 5670} C_VEL
LIN {X 0,Y 497.196,Z 855.945,A -85,B 0,C 180,E1 5673.48,E2 5673.48} C_VEL
LIN {X 0,Y 497.347,Z 849.599,A -85,B 0,C 180,E1 5677.848,E2 5677.848} C_VEL
LIN {X 0,Y 497.73,Z 838.031,A -85,B 0,C 180,E1 5682.254,E2 5682.254} C_VEL
LIN {X 0,Y 498.699,Z 820.515,A -85,B 0,C 180,E1 5686.708,E2 5686.708} C_VEL
LIN {X 0,Y 500.283,Z 797.892,A -85,B 0,C 180,E1 5690.876,E2 5690.876} C_VEL
LIN {X 0,Y 502.704,Z 770.161,A -85,B 0,C 180,E1 5694.706,E2 5694.706} C_VEL
LIN {X 0,Y 505.585,Z 738.41,A -85,B 0,C 180,E1 5698.022,E2 5698.022} C_VEL
LIN {X 0,Y 508.63,Z 703.472,A -85,B 0,C 180,E1 5700.741,E2 5700.741} C_VEL
LIN {X 0,Y 511.454,Z 665.342,A -85,B 0,C 180,E1 5702.859,E2 5702.859} C_VEL
LIN {X 0,Y 513.532,Z 626.934,A -85,B 0,C 180,E1 5704.255,E2 5704.255} C_VEL
LIN {X 0,Y 513.985,Z 586.523,A -85,B 0,C 180,E1 5705.083,E2 5705.083} C_VEL
LIN {X 0,Y 507.235,Z 575.263,A -85,B 0,C 180,E1 5705.752,E2 5705.752} C_VEL
LIN {X 0,Y 499.84,Z 561.974,A -85,B 0,C 180,E1 5706.626,E2 5706.626} C_VEL
LIN {X 0,Y 496.549,Z 549.53,A -85,B 0,C 180,E1 5707.675,E2 5707.675} C_VEL
LIN {X 0,Y 496.335,Z 549.53,A -85,B 0,C 180,E1 5714.374,E2 5714.374} C_VEL
LIN {X 0,Y 496.392,Z 549.53,A -85,B 0,C 180,E1 5720.333,E2 5720.333} C_VEL
LIN {X 0,Y 496.366,Z 549.53,A -85,B 0,C 180,E1 5726.828,E2 5726.828} C_VEL
LIN {X 0,Y 496.441,Z 549.53,A -85,B 0,C 180,E1 5732.878,E2 5732.878} C_VEL
LIN {X 0,Y 496.686,Z 549.53,A -85,B 0,C 180,E1 5736.946,E2 5736.946} C_VEL
LIN {X 0,Y 501.105,Z 573.753,A -85,B 0,C 180,E1 5737.442,E2 5737.442} C_VEL
LIN {X 0,Y 501.109,Z 606.457,A -85,B 0,C 180,E1 5738.153,E2 5738.153} C_VEL
LIN {X 0,Y 500.644,Z 633.24,A -85,B 0,C 180,E1 5739.387,E2 5739.387} C_VEL
LIN {X 0,Y 499.956,Z 658.017,A -85,B 0,C 180,E1 5741.252,E2 5741.252} C_VEL
LIN {X 0,Y 499.228,Z 678.344,A -85,B 0,C 180,E1 5743.542,E2 5743.542} C_VEL
LIN {X 0,Y 498.584,Z 695.419,A -85,B 0,C 180,E1 5746.438,E2 5746.438} C_VEL
LIN {X 0,Y 498.151,Z 706.746,A -85,B 0,C 180,E1 5749.532,E2 5749.532} C_VEL
LIN {X 0,Y 497.915,Z 712.002,A -85,B 0,C 180,E1 5752.166,E2 5752.166} C_VEL
LIN {X 0,Y 497.899,Z 713.729,A -85,B 0,C 180,E1 5754.787,E2 5754.787} C_VEL
LIN {X 0,Y 497.944,Z 710.815,A -85,B 0,C 180,E1 5758.267,E2 5758.267} C_VEL
LIN {X 0,Y 498.164,Z 703.047,A -85,B 0,C 180,E1 5761.349,E2 5761.349} C_VEL
LIN {X 0,Y 498.567,Z 690.024,A -85,B 0,C 180,E1 5764.344,E2 5764.344} C_VEL
LIN {X 0,Y 499.3,Z 670.961,A -85,B 0,C 180,E1 5767.166,E2 5767.166} C_VEL
LIN {X 0,Y 500.176,Z 647.958,A -85,B 0,C 180,E1 5769.446,E2 5769.446} C_VEL
LIN {X 0,Y 500.881,Z 621.377,A -85,B 0,C 180,E1 5771.162,E2 5771.162} C_VEL
LIN {X 0,Y 501.466,Z 592.354,A -85,B 0,C 180,E1 5772.248,E2 5772.248} C_VEL
LIN {X 0,Y 500.665,Z 565.414,A -85,B 0,C 180,E1 5772.751,E2 5772.751} C_VEL
LIN {X 0,Y 497.005,Z 549.53,A -85,B 0,C 180,E1 5773.125,E2 5773.125} C_VEL
LIN {X 0,Y 496.704,Z 549.53,A -85,B 0,C 180,E1 5779.628,E2 5779.628} C_VEL
LIN {X 0,Y 496.543,Z 549.53,A -85,B 0,C 180,E1 5785.185,E2 5785.185} C_VEL
LIN {X 0,Y 496.354,Z 549.53,A -85,B 0,C 180,E1 5791.642,E2 5791.642} C_VEL
LIN {X 0,Y 496.231,Z 549.53,A -85,B 0,C 180,E1 5797.746,E2 5797.746} C_VEL
LIN {X 0,Y 496.285,Z 549.53,A -85,B 0,C 180,E1 5804.38,E2 5804.38} C_VEL
LIN {X 0,Y 496.347,Z 549.53,A -85,B 0,C 180,E1 5810.319,E2 5810.319} C_VEL
LIN {X 0,Y 496.339,Z 549.53,A -85,B 0,C 180,E1 5816.818,E2 5816.818} C_VEL
LIN {X 0,Y 496.516,Z 549.53,A -85,B 0,C 180,E1 5821.93,E2 5821.93} C_VEL
LIN {X 0,Y 509.284,Z 583.433,A -85,B 0,C 180,E1 5823.549,E2 5823.549} C_VEL
LIN {X 0,Y 507.56,Z 619.25,A -85,B 0,C 180,E1 5824.95,E2 5824.95} C_VEL
LIN {X 0,Y 505.218,Z 653.626,A -85,B 0,C 180,E1 5827.033,E2 5827.033} C_VEL
LIN {X 0,Y 502.789,Z 684.678,A -85,B 0,C 180,E1 5829.693,E2 5829.693} C_VEL
LIN {X 0,Y 500.439,Z 713.862,A -85,B 0,C 180,E1 5833.127,E2 5833.127} C_VEL
LIN {X 0,Y 498.808,Z 736.278,A -85,B 0,C 180,E1 5836.662,E2 5836.662} C_VEL
LIN {X 0,Y 497.889,Z 754.512,A -85,B 0,C 180,E1 5840.609,E2 5840.609} C_VEL
LIN {X 0,Y 497.429,Z 766.518,A -85,B 0,C 180,E1 5844.342,E2 5844.342} C_VEL
LIN {X 0,Y 497.286,Z 774.193,A -85,B 0,C 180,E1 5848.261,E2 5848.261} C_VEL
LIN {X 0,Y 497.219,Z 777.21,A -85,B 0,C 180,E1 5851.74,E2 5851.74} C_VEL
LIN {X 0,Y 497.234,Z 776.67,A -85,B 0,C 180,E1 5855.225,E2 5855.225} C_VEL
LIN {X 0,Y 497.379,Z 771.571,A -85,B 0,C 180,E1 5859.298,E2 5859.298} C_VEL
LIN {X 0,Y 497.652,Z 760.64,A -85,B 0,C 180,E1 5863.562,E2 5863.562} C_VEL
LIN {X 0,Y 498.433,Z 744.571,A -85,B 0,C 180,E1 5867.625,E2 5867.625} C_VEL
LIN {X 0,Y 499.916,Z 721.439,A -85,B 0,C 180,E1 5871.704,E2 5871.704} C_VEL
LIN {X 0,Y 501.919,Z 695.139,A -85,B 0,C 180,E1 5875.095,E2 5875.095} C_VEL
LIN {X 0,Y 504.209,Z 666.689,A -85,B 0,C 180,E1 5877.864,E2 5877.864} C_VEL
LIN {X 0,Y 506.535,Z 634.122,A -85,B 0,C 180,E1 5880.161,E2 5880.161} C_VEL
LIN {X 0,Y 508.583,Z 597.54,A -85,B 0,C 180,E1 5881.9,E2 5881.9} C_VEL
LIN {X 0,Y 508.589,Z 581.128,A -85,B 0,C 180,E1 5882.477,E2 5882.477} C_VEL
LIN {X 0,Y 496.657,Z 549.53,A -85,B 0,C 180,E1 5884.014,E2 5884.014} C_VEL
LIN {X 0,Y 496.332,Z 549.53,A -85,B 0,C 180,E1 5890.522,E2 5890.522} C_VEL
LIN {X 0,Y 496.28,Z 549.53,A -85,B 0,C 180,E1 5896.873,E2 5896.873} C_VEL
LIN {X 0,Y 496.489,Z 549.53,A -85,B 0,C 180,E1 5902.559,E2 5902.559} C_VEL
LIN {X 0,Y 496.49,Z 549.53,A -85,B 0,C 180,E1 5908.334,E2 5908.334} C_VEL
LIN {X 0,Y 496.453,Z 549.53,A -85,B 0,C 180,E1 5914.81,E2 5914.81} C_VEL
LIN {X 0,Y 496.657,Z 549.53,A -85,B 0,C 180,E1 5920.286,E2 5920.286} C_VEL
LIN {X 0,Y 500.562,Z 573.763,A -85,B 0,C 180,E1 5920.792,E2 5920.792} C_VEL
LIN {X 0,Y 500.4,Z 618.423,A -85,B 0,C 180,E1 5921.595,E2 5921.595} C_VEL
LIN {X 0,Y 499.972,Z 644.62,A -85,B 0,C 180,E1 5922.769,E2 5922.769} C_VEL
LIN {X 0,Y 499.335,Z 668.269,A -85,B 0,C 180,E1 5924.589,E2 5924.589} C_VEL
LIN {X 0,Y 498.677,Z 687.366,A -85,B 0,C 180,E1 5926.878,E2 5926.878} C_VEL
LIN {X 0,Y 498.336,Z 701.567,A -85,B 0,C 180,E1 5929.528,E2 5929.528} C_VEL
LIN {X 0,Y 498.039,Z 710.773,A -85,B 0,C 180,E1 5932.503,E2 5932.503} C_VEL
LIN {X 0,Y 497.964,Z 714.081,A -85,B 0,C 180,E1 5934.78,E2 5934.78} C_VEL
LIN {X 0,Y 497.976,Z 714.514,A -85,B 0,C 180,E1 5936.521,E2 5936.521} C_VEL
LIN {X 0,Y 498.092,Z 711.837,A -85,B 0,C 180,E1 5939.108,E2 5939.108} C_VEL
LIN {X 0,Y 498.373,Z 703.346,A -85,B 0,C 180,E1 5942.121,E2 5942.121} C_VEL
LIN {X 0,Y 498.827,Z 690.022,A -85,B 0,C 180,E1 5944.768,E2 5944.768} C_VEL
LIN {X 0,Y 499.417,Z 672.105,A -85,B 0,C 180,E1 5947.047,E2 5947.047} C_VEL
LIN {X 0,Y 500.003,Z 649.561,A -85,B 0,C 180,E1 5948.894,E2 5948.894} C_VEL
LIN {X 0,Y 500.434,Z 623.62,A -85,B 0,C 180,E1 5950.145,E2 5950.145} C_VEL
LIN {X 0,Y 500.432,Z 590.496,A -85,B 0,C 180,E1 5950.828,E2 5950.828} C_VEL
LIN {X 0,Y 499.514,Z 561.159,A -85,B 0,C 180,E1 5951.292,E2 5951.292} C_VEL
LIN {X 0,Y 496.982,Z 549.53,A -85,B 0,C 180,E1 5951.602,E2 5951.602} C_VEL
LIN {X 0,Y 496.683,Z 549.53,A -85,B 0,C 180,E1 5957.683,E2 5957.683} C_VEL
LIN {X 0,Y 496.492,Z 549.53,A -85,B 0,C 180,E1 5963.269,E2 5963.269} C_VEL
LIN {X 0,Y 496.357,Z 549.53,A -85,B 0,C 180,E1 5969.102,E2 5969.102} C_VEL
LIN {X 0,Y 496.331,Z 549.53,A -85,B 0,C 180,E1 5975.579,E2 5975.579} C_VEL
LIN {X 0,Y 492.327,Z 549.53,A -85,B 0,C 180,E1 5977.558,E2 5977.558} C_VEL
LIN {X 0,Y 488.414,Z 549.53,A -85,B 0,C 180,E1 5979.569,E2 5979.569} C_VEL
LIN {X 0,Y 488.425,Z 549.53,A -85,B 0,C 180,E1 5985.278,E2 5985.278} C_VEL
LIN {X 0,Y 488.52,Z 550.276,A -85,B 0,C 180,E1 5991.764,E2 5991.764} C_VEL
LIN {X 0,Y 492.247,Z 564.004,A -85,B 0,C 180,E1 5992.924,E2 5992.924} C_VEL
LIN {X 0,Y 500.961,Z 579.657,A -85,B 0,C 180,E1 5993.862,E2 5993.862} C_VEL
LIN {X 0,Y 507.387,Z 588.937,A -85,B 0,C 180,E1 5994.489,E2 5994.489} C_VEL
LIN {X 0,Y 506.373,Z 634.314,A -85,B 0,C 180,E1 5995.509,E2 5995.509} C_VEL
LIN {X 0,Y 504.171,Z 673.866,A -85,B 0,C 180,E1 5997.07,E2 5997.07} C_VEL
LIN {X 0,Y 501.192,Z 709.535,A -85,B 0,C 180,E1 5999.209,E2 5999.209} C_VEL
LIN {X 0,Y 497.76,Z 744.773,A -85,B 0,C 180,E1 6002.137,E2 6002.137} C_VEL
LIN {X 0,Y 494.681,Z 776.028,A -85,B 0,C 180,E1 6005.631,E2 6005.631} C_VEL
LIN {X 0,Y 492.345,Z 801.504,A -85,B 0,C 180,E1 6009.383,E2 6009.383} C_VEL
LIN {X 0,Y 490.632,Z 822.692,A -85,B 0,C 180,E1 6013.501,E2 6013.501} C_VEL
LIN {X 0,Y 489.739,Z 839.42,A -85,B 0,C 180,E1 6017.994,E2 6017.994} C_VEL
LIN {X 0,Y 489.451,Z 849.597,A -85,B 0,C 180,E1 6022.024,E2 6022.024} C_VEL
LIN {X 0,Y 489.284,Z 855.945,A -85,B 0,C 180,E1 6026.463,E2 6026.463} C_VEL
LIN {X 0,Y 489.325,Z 857.5,A -85,B 0,C 180,E1 6030,E2 6030} C_VEL
LIN {X 0,Y 489.294,Z 855.945,A -85,B 0,C 180,E1 6033.536,E2 6033.536} C_VEL
LIN {X 0,Y 489.474,Z 849.599,A -85,B 0,C 180,E1 6037.975,E2 6037.975} C_VEL
LIN {X 0,Y 489.887,Z 838.031,A -85,B 0,C 180,E1 6042.453,E2 6042.453} C_VEL
LIN {X 0,Y 490.905,Z 820.839,A -85,B 0,C 180,E1 6046.91,E2 6046.91} C_VEL
LIN {X 0,Y 492.717,Z 797.697,A -85,B 0,C 180,E1 6051.244,E2 6051.244} C_VEL
LIN {X 0,Y 495.265,Z 770.775,A -85,B 0,C 180,E1 6055.025,E2 6055.025} C_VEL
LIN {X 0,Y 498.377,Z 738.667,A -85,B 0,C 180,E1 6058.438,E2 6058.438} C_VEL
LIN {X 0,Y 501.763,Z 703.11,A -85,B 0,C 180,E1 6061.234,E2 6061.234} C_VEL
LIN {X 0,Y 504.567,Z 666.944,A -85,B 0,C 180,E1 6063.262,E2 6063.262} C_VEL
LIN {X 0,Y 506.786,Z 626.334,A -85,B 0,C 180,E1 6064.724,E2 6064.724} C_VEL
LIN {X 0,Y 507.12,Z 588.801,A -85,B 0,C 180,E1 6065.537,E2 6065.537} C_VEL
LIN {X 0,Y 499.953,Z 577.705,A -85,B 0,C 180,E1 6066.255,E2 6066.255} C_VEL
LIN {X 0,Y 491.044,Z 558.665,A -85,B 0,C 180,E1 6067.379,E2 6067.379} C_VEL
LIN {X 0,Y 488.601,Z 549.53,A -85,B 0,C 180,E1 6068.248,E2 6068.248} C_VEL
LIN {X 0,Y 488.433,Z 549.53,A -85,B 0,C 180,E1 6075.288,E2 6075.288} C_VEL
LIN {X 0,Y 488.487,Z 549.53,A -85,B 0,C 180,E1 6081.847,E2 6081.847} C_VEL
LIN {X 0,Y 488.44,Z 549.53,A -85,B 0,C 180,E1 6088.322,E2 6088.322} C_VEL
LIN {X 0,Y 488.558,Z 549.53,A -85,B 0,C 180,E1 6094.383,E2 6094.383} C_VEL
LIN {X 0,Y 488.732,Z 549.53,A -85,B 0,C 180,E1 6096.669,E2 6096.669} C_VEL
LIN {X 0,Y 493.471,Z 572.27,A -85,B 0,C 180,E1 6097.189,E2 6097.189} C_VEL
LIN {X 0,Y 493.517,Z 605.325,A -85,B 0,C 180,E1 6097.868,E2 6097.868} C_VEL
LIN {X 0,Y 493.051,Z 633.332,A -85,B 0,C 180,E1 6099.124,E2 6099.124} C_VEL
LIN {X 0,Y 492.373,Z 658.496,A -85,B 0,C 180,E1 6101.001,E2 6101.001} C_VEL
LIN {X 0,Y 491.594,Z 678.848,A -85,B 0,C 180,E1 6103.279,E2 6103.279} C_VEL
LIN {X 0,Y 490.929,Z 695.254,A -85,B 0,C 180,E1 6105.996,E2 6105.996} C_VEL
LIN {X 0,Y 490.505,Z 706.609,A -85,B 0,C 180,E1 6108.918,E2 6108.918} C_VEL
LIN {X 0,Y 490.152,Z 713.27,A -85,B 0,C 180,E1 6112.041,E2 6112.041} C_VEL
LIN {X 0,Y 490.132,Z 715.064,A -85,B 0,C 180,E1 6114.704,E2 6114.704} C_VEL
LIN {X 0,Y 490.186,Z 712.233,A -85,B 0,C 180,E1 6118.24,E2 6118.24} C_VEL
LIN {X 0,Y 490.404,Z 704.491,A -85,B 0,C 180,E1 6121.37,E2 6121.37} C_VEL
LIN {X 0,Y 490.831,Z 691.471,A -85,B 0,C 180,E1 6124.412,E2 6124.412} C_VEL
LIN {X 0,Y 491.503,Z 674.267,A -85,B 0,C 180,E1 6127.058,E2 6127.058} C_VEL
LIN {X 0,Y 492.422,Z 650.796,A -85,B 0,C 180,E1 6129.485,E2 6129.485} C_VEL
LIN {X 0,Y 493.195,Z 624.695,A -85,B 0,C 180,E1 6131.255,E2 6131.255} C_VEL
LIN {X 0,Y 493.838,Z 594.763,A -85,B 0,C 180,E1 6132.433,E2 6132.433} C_VEL
LIN {X 0,Y 493.004,Z 566.309,A -85,B 0,C 180,E1 6132.985,E2 6132.985} C_VEL
LIN {X 0,Y 489.087,Z 549.53,A -85,B 0,C 180,E1 6133.42,E2 6133.42} C_VEL
LIN {X 0,Y 488.792,Z 549.53,A -85,B 0,C 180,E1 6139.857,E2 6139.857} C_VEL
LIN {X 0,Y 488.571,Z 549.53,A -85,B 0,C 180,E1 6145.625,E2 6145.625} C_VEL
LIN {X 0,Y 488.45,Z 549.53,A -85,B 0,C 180,E1 6151.687,E2 6151.687} C_VEL
LIN {X 0,Y 488.312,Z 549.53,A -85,B 0,C 180,E1 6158.18,E2 6158.18} C_VEL
LIN {X 0,Y 488.385,Z 549.53,A -85,B 0,C 180,E1 6164.706,E2 6164.706} C_VEL
LIN {X 0,Y 488.414,Z 549.53,A -85,B 0,C 180,E1 6170.577,E2 6170.577} C_VEL
LIN {X 0,Y 488.419,Z 549.53,A -85,B 0,C 180,E1 6176.54,E2 6176.54} C_VEL
LIN {X 0,Y 488.584,Z 550.196,A -85,B 0,C 180,E1 6181.41,E2 6181.41} C_VEL
LIN {X 0,Y 502.275,Z 584.851,A -85,B 0,C 180,E1 6183.162,E2 6183.162} C_VEL
LIN {X 0,Y 500.475,Z 619.532,A -85,B 0,C 180,E1 6184.546,E2 6184.546} C_VEL
LIN {X 0,Y 497.993,Z 654.496,A -85,B 0,C 180,E1 6186.681,E2 6186.681} C_VEL
LIN {X 0,Y 495.537,Z 684.37,A -85,B 0,C 180,E1 6189.265,E2 6189.265} C_VEL
LIN {X 0,Y 493.119,Z 711.202,A -85,B 0,C 180,E1 6192.409,E2 6192.409} C_VEL
LIN {X 0,Y 491.182,Z 735.365,A -85,B 0,C 180,E1 6196.225,E2 6196.225} C_VEL
LIN {X 0,Y 490.119,Z 753.561,A -85,B 0,C 180,E1 6200.17,E2 6200.17} C_VEL
LIN {X 0,Y 489.562,Z 766.63,A -85,B 0,C 180,E1 6204.25,E2 6204.25} C_VEL
LIN {X 0,Y 489.388,Z 774.254,A -85,B 0,C 180,E1 6208.233,E2 6208.233} C_VEL
LIN {X 0,Y 489.316,Z 777.221,A -85,B 0,C 180,E1 6211.768,E2 6211.768} C_VEL
LIN {X 0,Y 489.325,Z 776.635,A -85,B 0,C 180,E1 6215.309,E2 6215.309} C_VEL
LIN {X 0,Y 489.478,Z 771.596,A -85,B 0,C 180,E1 6219.387,E2 6219.387} C_VEL
LIN {X 0,Y 489.818,Z 760.52,A -85,B 0,C 180,E1 6223.77,E2 6223.77} C_VEL
LIN {X 0,Y 490.647,Z 744.328,A -85,B 0,C 180,E1 6227.914,E2 6227.914} C_VEL
LIN {X 0,Y 492.368,Z 720.046,A -85,B 0,C 180,E1 6232.242,E2 6232.242} C_VEL
LIN {X 0,Y 494.722,Z 692.791,A -85,B 0,C 180,E1 6235.76,E2 6235.76} C_VEL
LIN {X 0,Y 497.455,Z 661.818,A -85,B 0,C 180,E1 6238.672,E2 6238.672} C_VEL
LIN {X 0,Y 499.869,Z 628.733,A -85,B 0,C 180,E1 6240.881,E2 6240.881} C_VEL
LIN {X 0,Y 501.809,Z 592.342,A -85,B 0,C 180,E1 6242.515,E2 6242.515} C_VEL
LIN {X 0,Y 501.242,Z 582.253,A -85,B 0,C 180,E1 6242.897,E2 6242.897} C_VEL
LIN {X 0,Y 488.739,Z 549.53,A -85,B 0,C 180,E1 6244.597,E2 6244.597} C_VEL
LIN {X 0,Y 488.436,Z 549.53,A -85,B 0,C 180,E1 6250.456,E2 6250.456} C_VEL
LIN {X 0,Y 488.378,Z 549.53,A -85,B 0,C 180,E1 6257.169,E2 6257.169} C_VEL
LIN {X 0,Y 488.569,Z 549.53,A -85,B 0,C 180,E1 6263.431,E2 6263.431} C_VEL
LIN {X 0,Y 488.59,Z 549.53,A -85,B 0,C 180,E1 6268.324,E2 6268.324} C_VEL
LIN {X 0,Y 488.49,Z 549.53,A -85,B 0,C 180,E1 6274.37,E2 6274.37} C_VEL
LIN {X 0,Y 488.715,Z 549.53,A -85,B 0,C 180,E1 6280.051,E2 6280.051} C_VEL
LIN {X 0,Y 492.904,Z 574.491,A -85,B 0,C 180,E1 6280.58,E2 6280.58} C_VEL
LIN {X 0,Y 492.731,Z 618.32,A -85,B 0,C 180,E1 6281.365,E2 6281.365} C_VEL
LIN {X 0,Y 492.313,Z 644.098,A -85,B 0,C 180,E1 6282.492,E2 6282.492} C_VEL
LIN {X 0,Y 491.708,Z 667.494,A -85,B 0,C 180,E1 6284.251,E2 6284.251} C_VEL
LIN {X 0,Y 491.057,Z 686.382,A -85,B 0,C 180,E1 6286.444,E2 6286.444} C_VEL
LIN {X 0,Y 490.642,Z 700.484,A -85,B 0,C 180,E1 6288.913,E2 6288.913} C_VEL
LIN {X 0,Y 490.283,Z 711.161,A -85,B 0,C 180,E1 6292.035,E2 6292.035} C_VEL
LIN {X 0,Y 490.206,Z 715.322,A -85,B 0,C 180,E1 6294.697,E2 6294.697} C_VEL
LIN {X 0,Y 490.211,Z 715.829,A -85,B 0,C 180,E1 6296.466,E2 6296.466} C_VEL
LIN {X 0,Y 490.331,Z 713.263,A -85,B 0,C 180,E1 6299.094,E2 6299.094} C_VEL
LIN {X 0,Y 490.62,Z 704.884,A -85,B 0,C 180,E1 6302.155,E2 6302.155} C_VEL
LIN {X 0,Y 491.127,Z 691.644,A -85,B 0,C 180,E1 6304.843,E2 6304.843} C_VEL
LIN {X 0,Y 491.732,Z 673.819,A -85,B 0,C 180,E1 6307.158,E2 6307.158} C_VEL
LIN {X 0,Y 492.337,Z 651.379,A -85,B 0,C 180,E1 6309.034,E2 6309.034} C_VEL
LIN {X 0,Y 492.718,Z 625.731,A -85,B 0,C 180,E1 6310.306,E2 6310.306} C_VEL
LIN {X 0,Y 492.759,Z 593.964,A -85,B 0,C 180,E1 6310.994,E2 6310.994} C_VEL
LIN {X 0,Y 492.15,Z 563.51,A -85,B 0,C 180,E1 6311.479,E2 6311.479} C_VEL
LIN {X 0,Y 489.023,Z 549.53,A -85,B 0,C 180,E1 6311.819,E2 6311.819} C_VEL
LIN {X 0,Y 488.742,Z 549.53,A -85,B 0,C 180,E1 6317.98,E2 6317.98} C_VEL
LIN {X 0,Y 488.57,Z 549.53,A -85,B 0,C 180,E1 6323.669,E2 6323.669} C_VEL
LIN {X 0,Y 488.357,Z 549.53,A -85,B 0,C 180,E1 6330.084,E2 6330.084} C_VEL
LIN {X 0,Y 488.394,Z 549.53,A -85,B 0,C 180,E1 6335.944,E2 6335.944} C_VEL
LIN {X 0,Y 488.414,Z 549.53,A -85,B 0,C 180,E1 6339.569,E2 6339.569} C_VEL
LIN {X 0,Y 485.813,Z 549.53,A -85,B 0,C 180,E1 6341.075,E2 6341.075} C_VEL
LIN {X 0,Y 480.507,Z 549.53,A -85,B 0,C 180,E1 6343.334,E2 6343.334} C_VEL
LIN {X 0,Y 480.45,Z 549.53,A -85,B 0,C 180,E1 6343.595,E2 6343.595} C_VEL
LIN {X 0,Y 480.42,Z 549.53,A -85,B 0,C 180,E1 6348.919,E2 6348.919} C_VEL
LIN {X 0,Y 480.538,Z 550.006,A -85,B 0,C 180,E1 6351.256,E2 6351.256} C_VEL
LIN {X 0,Y 483.559,Z 560.744,A -85,B 0,C 180,E1 6352.165,E2 6352.165} C_VEL
LIN {X 0,Y 494.033,Z 582.814,A -85,B 0,C 180,E1 6353.388,E2 6353.388} C_VEL
LIN {X 0,Y 500.869,Z 591.84,A -85,B 0,C 180,E1 6354.06,E2 6354.06} C_VEL
LIN {X 0,Y 499.44,Z 635.85,A -85,B 0,C 180,E1 6355.107,E2 6355.107} C_VEL
LIN {X 0,Y 497.011,Z 675.621,A -85,B 0,C 180,E1 6356.736,E2 6356.736} C_VEL
LIN {X 0,Y 493.968,Z 712.701,A -85,B 0,C 180,E1 6358.967,E2 6358.967} C_VEL
LIN {X 0,Y 490.518,Z 745.799,A -85,B 0,C 180,E1 6361.797,E2 6361.797} C_VEL
LIN {X 0,Y 487.238,Z 776.376,A -85,B 0,C 180,E1 6365.282,E2 6365.282} C_VEL
LIN {X 0,Y 484.656,Z 802.407,A -85,B 0,C 180,E1 6369.201,E2 6369.201} C_VEL
LIN {X 0,Y 482.866,Z 822.869,A -85,B 0,C 180,E1 6373.27,E2 6373.27} C_VEL
LIN {X 0,Y 481.906,Z 839.422,A -85,B 0,C 180,E1 6377.796,E2 6377.796} C_VEL
LIN {X 0,Y 481.557,Z 849.596,A -85,B 0,C 180,E1 6381.892,E2 6381.892} C_VEL
LIN {X 0,Y 481.385,Z 855.944,A -85,B 0,C 180,E1 6386.405,E2 6386.405} C_VEL
LIN {X 0,Y 481.431,Z 857.5,A -85,B 0,C 180,E1 6390,E2 6390} C_VEL
LIN {X 0,Y 481.397,Z 855.944,A -85,B 0,C 180,E1 6393.594,E2 6393.594} C_VEL
LIN {X 0,Y 481.583,Z 849.598,A -85,B 0,C 180,E1 6398.107,E2 6398.107} C_VEL
LIN {X 0,Y 482.127,Z 836.87,A -85,B 0,C 180,E1 6403.019,E2 6403.019} C_VEL
LIN {X 0,Y 483.258,Z 819.42,A -85,B 0,C 180,E1 6407.5,E2 6407.5} C_VEL
LIN {X 0,Y 485.308,Z 795.751,A -85,B 0,C 180,E1 6411.911,E2 6411.911} C_VEL
LIN {X 0,Y 488.21,Z 767.337,A -85,B 0,C 180,E1 6415.857,E2 6415.857} C_VEL
LIN {X 0,Y 491.71,Z 734.703,A -85,B 0,C 180,E1 6419.249,E2 6419.249} C_VEL
LIN {X 0,Y 494.843,Z 702.275,A -85,B 0,C 180,E1 6421.741,E2 6421.741} C_VEL
LIN {X 0,Y 497.867,Z 663.384,A -85,B 0,C 180,E1 6423.845,E2 6423.845} C_VEL
LIN {X 0,Y 500.082,Z 624.407,A -85,B 0,C 180,E1 6425.239,E2 6425.239} C_VEL
LIN {X 0,Y 500.541,Z 591.439,A -85,B 0,C 180,E1 6425.981,E2 6425.981} C_VEL
LIN {X 0,Y 488.114,Z 570.777,A -85,B 0,C 180,E1 6427.302,E2 6427.302} C_VEL
LIN {X 0,Y 482.122,Z 555.231,A -85,B 0,C 180,E1 6428.182,E2 6428.182} C_VEL
LIN {X 0,Y 480.614,Z 549.53,A -85,B 0,C 180,E1 6428.738,E2 6428.738} C_VEL
LIN {X 0,Y 480.46,Z 549.53,A -85,B 0,C 180,E1 6433.754,E2 6433.754} C_VEL
LIN {X 0,Y 480.524,Z 549.53,A -85,B 0,C 180,E1 6438.917,E2 6438.917} C_VEL
LIN {X 0,Y 480.496,Z 549.53,A -85,B 0,C 180,E1 6444.748,E2 6444.748} C_VEL
LIN {X 0,Y 480.524,Z 549.53,A -85,B 0,C 180,E1 6449.842,E2 6449.842} C_VEL
LIN {X 0,Y 480.805,Z 549.53,A -85,B 0,C 180,E1 6456.37,E2 6456.37} C_VEL
LIN {X 0,Y 485.891,Z 575.928,A -85,B 0,C 180,E1 6457.004,E2 6457.004} C_VEL
LIN {X 0,Y 485.92,Z 608.281,A -85,B 0,C 180,E1 6457.71,E2 6457.71} C_VEL
LIN {X 0,Y 485.449,Z 636.564,A -85,B 0,C 180,E1 6459.036,E2 6459.036} C_VEL
LIN {X 0,Y 484.653,Z 662.195,A -85,B 0,C 180,E1 6461.04,E2 6461.04} C_VEL
LIN {X 0,Y 483.85,Z 682.72,A -85,B 0,C 180,E1 6463.476,E2 6463.476} C_VEL
LIN {X 0,Y 483.111,Z 699.296,A -85,B 0,C 180,E1 6466.456,E2 6466.456} C_VEL
LIN {X 0,Y 482.696,Z 708.989,A -85,B 0,C 180,E1 6469.193,E2 6469.193} C_VEL
LIN {X 0,Y 482.4,Z 714.545,A -85,B 0,C 180,E1 6471.912,E2 6471.912} C_VEL
LIN {X 0,Y 482.355,Z 716.408,A -85,B 0,C 180,E1 6474.619,E2 6474.619} C_VEL
LIN {X 0,Y 482.427,Z 713.648,A -85,B 0,C 180,E1 6478.212,E2 6478.212} C_VEL
LIN {X 0,Y 482.632,Z 706.076,A -85,B 0,C 180,E1 6481.348,E2 6481.348} C_VEL
LIN {X 0,Y 483.095,Z 692.915,A -85,B 0,C 180,E1 6484.483,E2 6484.483} C_VEL
LIN {X 0,Y 483.801,Z 675.717,A -85,B 0,C 180,E1 6487.171,E2 6487.171} C_VEL
LIN {X 0,Y 484.718,Z 653.566,A -85,B 0,C 180,E1 6489.524,E2 6489.524} C_VEL
LIN {X 0,Y 485.523,Z 627.393,A -85,B 0,C 180,E1 6491.373,E2 6491.373} C_VEL
LIN {X 0,Y 486.138,Z 599.428,A -85,B 0,C 180,E1 6492.554,E2 6492.554} C_VEL
LIN {X 0,Y 485.478,Z 567.766,A -85,B 0,C 180,E1 6493.212,E2 6493.212} C_VEL
LIN {X 0,Y 481.139,Z 549.53,A -85,B 0,C 180,E1 6493.705,E2 6493.705} C_VEL
LIN {X 0,Y 480.837,Z 549.53,A -85,B 0,C 180,E1 6500.199,E2 6500.199} C_VEL
LIN {X 0,Y 480.657,Z 549.53,A -85,B 0,C 180,E1 6506.079,E2 6506.079} C_VEL
LIN {X 0,Y 480.529,Z 549.53,A -85,B 0,C 180,E1 6512.271,E2 6512.271} C_VEL
LIN {X 0,Y 480.379,Z 549.53,A -85,B 0,C 180,E1 6518.928,E2 6518.928} C_VEL
LIN {X 0,Y 480.436,Z 549.53,A -85,B 0,C 180,E1 6523.74,E2 6523.74} C_VEL
LIN {X 0,Y 480.491,Z 549.53,A -85,B 0,C 180,E1 6528.922,E2 6528.922} C_VEL
LIN {X 0,Y 480.43,Z 549.53,A -85,B 0,C 180,E1 6534.759,E2 6534.759} C_VEL
LIN {X 0,Y 480.617,Z 549.53,A -85,B 0,C 180,E1 6540.831,E2 6540.831} C_VEL
LIN {X 0,Y 495.23,Z 587.24,A -85,B 0,C 180,E1 6542.799,E2 6542.799} C_VEL
LIN {X 0,Y 493.275,Z 622.788,A -85,B 0,C 180,E1 6544.276,E2 6544.276} C_VEL
LIN {X 0,Y 490.628,Z 656.715,A -85,B 0,C 180,E1 6546.43,E2 6546.43} C_VEL
LIN {X 0,Y 487.921,Z 687.341,A -85,B 0,C 180,E1 6549.164,E2 6549.164} C_VEL
LIN {X 0,Y 485.3,Z 715.307,A -85,B 0,C 180,E1 6552.584,E2 6552.584} C_VEL
LIN {X 0,Y 483.275,Z 738.19,A -85,B 0,C 180,E1 6556.455,E2 6556.455} C_VEL
LIN {X 0,Y 482.205,Z 755.666,A -85,B 0,C 180,E1 6560.503,E2 6560.503} C_VEL
LIN {X 0,Y 481.652,Z 767.773,A -85,B 0,C 180,E1 6564.607,E2 6564.607} C_VEL
LIN {X 0,Y 481.504,Z 774.314,A -85,B 0,C 180,E1 6568.204,E2 6568.204} C_VEL
LIN {X 0,Y 481.437,Z 777.232,A -85,B 0,C 180,E1 6571.797,E2 6571.797} C_VEL
LIN {X 0,Y 481.417,Z 776.6,A -85,B 0,C 180,E1 6575.397,E2 6575.397} C_VEL
LIN {X 0,Y 481.577,Z 771.513,A -85,B 0,C 180,E1 6579.542,E2 6579.542} C_VEL
LIN {X 0,Y 481.947,Z 760.667,A -85,B 0,C 180,E1 6583.9,E2 6583.9} C_VEL
LIN {X 0,Y 482.906,Z 744.155,A -85,B 0,C 180,E1 6588.212,E2 6588.212} C_VEL
LIN {X 0,Y 484.691,Z 721.853,A -85,B 0,C 180,E1 6592.346,E2 6592.346} C_VEL
LIN {X 0,Y 487.09,Z 696.81,A -85,B 0,C 180,E1 6595.707,E2 6595.707} C_VEL
LIN {X 0,Y 489.753,Z 667.122,A -85,B 0,C 180,E1 6598.648,E2 6598.648} C_VEL
LIN {X 0,Y 492.424,Z 634.201,A -85,B 0,C 180,E1 6601.001,E2 6601.001} C_VEL
LIN {X 0,Y 494.554,Z 598.368,A -85,B 0,C 180,E1 6602.727,E2 6602.727} C_VEL
LIN {X 0,Y 494.448,Z 585.141,A -85,B 0,C 180,E1 6603.227,E2 6603.227} C_VEL
LIN {X 0,Y 480.803,Z 549.53,A -85,B 0,C 180,E1 6605.092,E2 6605.092} C_VEL
LIN {X 0,Y 480.478,Z 549.53,A -85,B 0,C 180,E1 6611.271,E2 6611.271} C_VEL
LIN {X 0,Y 480.412,Z 549.53,A -85,B 0,C 180,E1 6616.281,E2 6616.281} C_VEL
LIN {X 0,Y 480.629,Z 549.53,A -85,B 0,C 180,E1 6621.721,E2 6621.721} C_VEL
LIN {X 0,Y 480.666,Z 549.53,A -85,B 0,C 180,E1 6627.967,E2 6627.967} C_VEL
LIN {X 0,Y 480.569,Z 549.53,A -85,B 0,C 180,E1 6633.916,E2 6633.916} C_VEL
LIN {X 0,Y 480.766,Z 549.53,A -85,B 0,C 180,E1 6639.797,E2 6639.797} C_VEL
LIN {X 0,Y 484.998,Z 573.041,A -85,B 0,C 180,E1 6640.321,E2 6640.321} C_VEL
LIN {X 0,Y 485.077,Z 619.207,A -85,B 0,C 180,E1 6641.161,E2 6641.161} C_VEL
LIN {X 0,Y 484.652,Z 645.404,A -85,B 0,C 180,E1 6642.323,E2 6642.323} C_VEL
LIN {X 0,Y 483.951,Z 669.768,A -85,B 0,C 180,E1 6644.204,E2 6644.204} C_VEL
LIN {X 0,Y 483.265,Z 688.495,A -85,B 0,C 180,E1 6646.452,E2 6646.452} C_VEL
LIN {X 0,Y 482.861,Z 703.28,A -85,B 0,C 180,E1 6649.188,E2 6649.188} C_VEL
LIN {X 0,Y 482.526,Z 712.227,A -85,B 0,C 180,E1 6651.906,E2 6651.906} C_VEL
LIN {X 0,Y 482.426,Z 716.561,A -85,B 0,C 180,E1 6654.611,E2 6654.611} C_VEL
LIN {X 0,Y 482.43,Z 717.148,A -85,B 0,C 180,E1 6656.409,E2 6656.409} C_VEL
LIN {X 0,Y 482.561,Z 714.659,A -85,B 0,C 180,E1 6659.1,E2 6659.1} C_VEL
LIN {X 0,Y 482.893,Z 706.254,A -85,B 0,C 180,E1 6662.235,E2 6662.235} C_VEL
LIN {X 0,Y 483.417,Z 693.276,A -85,B 0,C 180,E1 6664.92,E2 6664.92} C_VEL
LIN {X 0,Y 484.066,Z 675.559,A -85,B 0,C 180,E1 6667.272,E2 6667.272} C_VEL
LIN {X 0,Y 484.681,Z 653.271,A -85,B 0,C 180,E1 6669.177,E2 6669.177} C_VEL
LIN {X 0,Y 485.079,Z 627.921,A -85,B 0,C 180,E1 6670.47,E2 6670.47} C_VEL
LIN {X 0,Y 485.095,Z 597.206,A -85,B 0,C 180,E1 6671.17,E2 6671.17} C_VEL
LIN {X 0,Y 484.39,Z 564.098,A -85,B 0,C 180,E1 6671.712,E2 6671.712} C_VEL
LIN {X 0,Y 481.079,Z 549.53,A -85,B 0,C 180,E1 6672.123,E2 6672.123} C_VEL
LIN {X 0,Y 480.802,Z 549.53,A -85,B 0,C 180,E1 6678.287,E2 6678.287} C_VEL
LIN {X 0,Y 480.611,Z 549.53,A -85,B 0,C 180,E1 6684.406,E2 6684.406} C_VEL
LIN {X 0,Y 480.46,Z 549.53,A -85,B 0,C 180,E1 6690.163,E2 6690.163} C_VEL
LIN {X 0,Y 480.523,Z 549.53,A -85,B 0,C 180,E1 6696.627,E2 6696.627} C_VEL
LIN {X 0,Y 480.491,Z 549.53,A -85,B 0,C 180,E1 6701.258,E2 6701.258} C_VEL
LIN {X 0,Y 480.45,Z 549.53,A -85,B 0,C 180,E1 6703.595,E2 6703.595} C_VEL
LIN {X 0,Y 478.001,Z 549.53,A -85,B 0,C 180,E1 6705.128,E2 6705.128} C_VEL
LIN {X 0,Y 472.526,Z 549.53,A -85,B 0,C 180,E1 6707.428,E2 6707.428} C_VEL
LIN {X 0,Y 472.426,Z 549.53,A -85,B 0,C 180,E1 6707.694,E2 6707.694} C_VEL
LIN {X 0,Y 472.585,Z 549.764,A -85,B 0,C 180,E1 6710.731,E2 6710.731} C_VEL
LIN {X 0,Y 475.25,Z 558.691,A -85,B 0,C 180,E1 6711.425,E2 6711.425} C_VEL
LIN {X 0,Y 487.518,Z 586.094,A -85,B 0,C 180,E1 6712.934,E2 6712.934} C_VEL
LIN {X 0,Y 494.304,Z 594.899,A -85,B 0,C 180,E1 6713.629,E2 6713.629} C_VEL
LIN {X 0,Y 492.566,Z 636.597,A -85,B 0,C 180,E1 6714.668,E2 6714.668} C_VEL
LIN {X 0,Y 489.957,Z 675.964,A -85,B 0,C 180,E1 6716.327,E2 6716.327} C_VEL
LIN {X 0,Y 486.739,Z 712.663,A -85,B 0,C 180,E1 6718.568,E2 6718.568} C_VEL
LIN {X 0,Y 483.303,Z 746.501,A -85,B 0,C 180,E1 6721.414,E2 6721.414} C_VEL
LIN {X 0,Y 479.891,Z 776.376,A -85,B 0,C 180,E1 6724.877,E2 6724.877} C_VEL
LIN {X 0,Y 477.076,Z 802.408,A -85,B 0,C 180,E1 6728.854,E2 6728.854} C_VEL
LIN {X 0,Y 475.119,Z 823.242,A -85,B 0,C 180,E1 6733.078,E2 6733.078} C_VEL
LIN {X 0,Y 474.048,Z 839.423,A -85,B 0,C 180,E1 6737.59,E2 6737.59} C_VEL
LIN {X 0,Y 473.676,Z 849.624,A -85,B 0,C 180,E1 6741.771,E2 6741.771} C_VEL
LIN {X 0,Y 473.48,Z 855.943,A -85,B 0,C 180,E1 6746.345,E2 6746.345} C_VEL
LIN {X 0,Y 473.531,Z 857.5,A -85,B 0,C 180,E1 6750,E2 6750} C_VEL
LIN {X 0,Y 473.494,Z 855.943,A -85,B 0,C 180,E1 6753.655,E2 6753.655} C_VEL
LIN {X 0,Y 473.702,Z 849.623,A -85,B 0,C 180,E1 6758.229,E2 6758.229} C_VEL
LIN {X 0,Y 474.295,Z 837.004,A -85,B 0,C 180,E1 6763.195,E2 6763.195} C_VEL
LIN {X 0,Y 475.555,Z 819.188,A -85,B 0,C 180,E1 6767.846,E2 6767.846} C_VEL
LIN {X 0,Y 477.754,Z 795.75,A -85,B 0,C 180,E1 6772.276,E2 6772.276} C_VEL
LIN {X 0,Y 480.878,Z 767.723,A -85,B 0,C 180,E1 6776.231,E2 6776.231} C_VEL
LIN {X 0,Y 484.26,Z 737.472,A -85,B 0,C 180,E1 6779.437,E2 6779.437} C_VEL
LIN {X 0,Y 487.667,Z 702.531,A -85,B 0,C 180,E1 6782.134,E2 6782.134} C_VEL
LIN {X 0,Y 490.915,Z 663.447,A -85,B 0,C 180,E1 6784.29,E2 6784.29} C_VEL
LIN {X 0,Y 493.404,Z 623.529,A -85,B 0,C 180,E1 6785.734,E2 6785.734} C_VEL
LIN {X 0,Y 494.038,Z 594.318,A -85,B 0,C 180,E1 6786.418,E2 6786.418} C_VEL
LIN {X 0,Y 483.225,Z 576.82,A -85,B 0,C 180,E1 6787.595,E2 6787.595} C_VEL
LIN {X 0,Y 472.978,Z 551.627,A -85,B 0,C 180,E1 6789.051,E2 6789.051} C_VEL
LIN {X 0,Y 472.64,Z 549.53,A -85,B 0,C 180,E1 6789.257,E2 6789.257} C_VEL
LIN {X 0,Y 472.495,Z 549.53,A -85,B 0,C 180,E1 6795.368,E2 6795.368} C_VEL
LIN {X 0,Y 472.572,Z 549.53,A -85,B 0,C 180,E1 6800.315,E2 6800.315} C_VEL
LIN {X 0,Y 472.545,Z 549.53,A -85,B 0,C 180,E1 6806.136,E2 6806.136} C_VEL
LIN {X 0,Y 472.612,Z 549.53,A -85,B 0,C 180,E1 6811.388,E2 6811.388} C_VEL
LIN {X 0,Y 472.864,Z 549.53,A -85,B 0,C 180,E1 6816.101,E2 6816.101} C_VEL
LIN {X 0,Y 478.235,Z 573.825,A -85,B 0,C 180,E1 6816.714,E2 6816.714} C_VEL
LIN {X 0,Y 478.337,Z 609.37,A -85,B 0,C 180,E1 6817.475,E2 6817.475} C_VEL
LIN {X 0,Y 477.883,Z 637.708,A -85,B 0,C 180,E1 6818.812,E2 6818.812} C_VEL
LIN {X 0,Y 477.057,Z 663.483,A -85,B 0,C 180,E1 6820.846,E2 6820.846} C_VEL
LIN {X 0,Y 476.239,Z 683.498,A -85,B 0,C 180,E1 6823.226,E2 6823.226} C_VEL
LIN {X 0,Y 475.474,Z 699.489,A -85,B 0,C 180,E1 6826.064,E2 6826.064} C_VEL
LIN {X 0,Y 474.972,Z 710.123,A -85,B 0,C 180,E1 6829.015,E2 6829.015} C_VEL
LIN {X 0,Y 474.639,Z 715.805,A -85,B 0,C 180,E1 6831.779,E2 6831.779} C_VEL
LIN {X 0,Y 474.588,Z 717.757,A -85,B 0,C 180,E1 6834.53,E2 6834.53} C_VEL
LIN {X 0,Y 474.667,Z 715.062,A -85,B 0,C 180,E1 6838.182,E2 6838.182} C_VEL
LIN {X 0,Y 474.868,Z 707.517,A -85,B 0,C 180,E1 6841.37,E2 6841.37} C_VEL
LIN {X 0,Y 475.342,Z 694.344,A -85,B 0,C 180,E1 6844.556,E2 6844.556} C_VEL
LIN {X 0,Y 476.101,Z 677.15,A -85,B 0,C 180,E1 6847.288,E2 6847.288} C_VEL
LIN {X 0,Y 477.036,Z 655.054,A -85,B 0,C 180,E1 6849.679,E2 6849.679} C_VEL
LIN {X 0,Y 477.892,Z 628.959,A -85,B 0,C 180,E1 6851.557,E2 6851.557} C_VEL
LIN {X 0,Y 478.537,Z 599.871,A -85,B 0,C 180,E1 6852.801,E2 6852.801} C_VEL
LIN {X 0,Y 478.155,Z 570.175,A -85,B 0,C 180,E1 6853.42,E2 6853.42} C_VEL
LIN {X 0,Y 473.19,Z 549.53,A -85,B 0,C 180,E1 6853.97,E2 6853.97} C_VEL
LIN {X 0,Y 472.891,Z 549.53,A -85,B 0,C 180,E1 6860.554,E2 6860.554} C_VEL
LIN {X 0,Y 472.698,Z 549.53,A -85,B 0,C 180,E1 6866.626,E2 6866.626} C_VEL
LIN {X 0,Y 472.536,Z 549.53,A -85,B 0,C 180,E1 6872.886,E2 6872.886} C_VEL
LIN {X 0,Y 472.46,Z 549.53,A -85,B 0,C 180,E1 6877.368,E2 6877.368} C_VEL
LIN {X 0,Y 472.441,Z 549.53,A -85,B 0,C 180,E1 6882.717,E2 6882.717} C_VEL
LIN {X 0,Y 472.477,Z 549.53,A -85,B 0,C 180,E1 6887.873,E2 6887.873} C_VEL
LIN {X 0,Y 472.577,Z 549.53,A -85,B 0,C 180,E1 6892.975,E2 6892.975} C_VEL
LIN {X 0,Y 472.649,Z 549.53,A -85,B 0,C 180,E1 6900.094,E2 6900.094} C_VEL
LIN {X 0,Y 472.997,Z 551.791,A -85,B 0,C 180,E1 6900.319,E2 6900.319} C_VEL
LIN {X 0,Y 488.19,Z 589.479,A -85,B 0,C 180,E1 6902.43,E2 6902.43} C_VEL
LIN {X 0,Y 486.083,Z 625.047,A -85,B 0,C 180,E1 6903.96,E2 6903.96} C_VEL
LIN {X 0,Y 483.246,Z 659.508,A -85,B 0,C 180,E1 6906.22,E2 6906.22} C_VEL
LIN {X 0,Y 480.35,Z 690.25,A -85,B 0,C 180,E1 6909.061,E2 6909.061} C_VEL
LIN {X 0,Y 477.623,Z 717.582,A -85,B 0,C 180,E1 6912.532,E2 6912.532} C_VEL
LIN {X 0,Y 475.594,Z 738.99,A -85,B 0,C 180,E1 6916.232,E2 6916.232} C_VEL
LIN {X 0,Y 474.386,Z 756.555,A -85,B 0,C 180,E1 6920.466,E2 6920.466} C_VEL
LIN {X 0,Y 473.806,Z 769.945,A -85,B 0,C 180,E1 6925.433,E2 6925.433} C_VEL
LIN {X 0,Y 473.69,Z 776.254,A -85,B 0,C 180,E1 6930,E2 6930} C_VEL
LIN {X 0,Y 473.539,Z 777.346,A -85,B 0,C 180,E1 6933.655,E2 6933.655} C_VEL
LIN {X 0,Y 473.631,Z 773.892,A -85,B 0,C 180,E1 6938.156,E2 6938.156} C_VEL
LIN {X 0,Y 473.901,Z 764.224,A -85,B 0,C 180,E1 6942.881,E2 6942.881} C_VEL
LIN {X 0,Y 474.838,Z 750.355,A -85,B 0,C 180,E1 6947.112,E2 6947.112} C_VEL
LIN {X 0,Y 476.267,Z 732.105,A -85,B 0,C 180,E1 6950.997,E2 6950.997} C_VEL
LIN {X 0,Y 478.602,Z 708.225,A -85,B 0,C 180,E1 6954.697,E2 6954.697} C_VEL
LIN {X 0,Y 481.366,Z 679.722,A -85,B 0,C 180,E1 6957.926,E2 6957.926} C_VEL
LIN {X 0,Y 484.221,Z 647.931,A -85,B 0,C 180,E1 6960.544,E2 6960.544} C_VEL
LIN {X 0,Y 486.832,Z 612.808,A -85,B 0,C 180,E1 6962.556,E2 6962.556} C_VEL
LIN {X 0,Y 487.469,Z 587.501,A -85,B 0,C 180,E1 6963.593,E2 6963.593} C_VEL
LIN {X 0,Y 472.828,Z 549.53,A -85,B 0,C 180,E1 6965.721,E2 6965.721} C_VEL
LIN {X 0,Y 472.455,Z 549.53,A -85,B 0,C 180,E1 6972.13,E2 6972.13} C_VEL
LIN {X 0,Y 472.459,Z 549.53,A -85,B 0,C 180,E1 6977.87,E2 6977.87} C_VEL
LIN {X 0,Y 472.747,Z 549.53,A -85,B 0,C 180,E1 6982.949,E2 6982.949} C_VEL
LIN {X 0,Y 472.706,Z 549.53,A -85,B 0,C 180,E1 6989.544,E2 6989.544} C_VEL
LIN {X 0,Y 472.668,Z 549.53,A -85,B 0,C 180,E1 6995.474,E2 6995.474} C_VEL
LIN {X 0,Y 472.821,Z 549.53,A -85,B 0,C 180,E1 6999.532,E2 6999.532} C_VEL
LIN {X 0,Y 477.365,Z 573.751,A -85,B 0,C 180,E1 7000.095,E2 7000.095} C_VEL
LIN {X 0,Y 477.439,Z 621.591,A -85,B 0,C 180,E1 7001.001,E2 7001.001} C_VEL
LIN {X 0,Y 476.957,Z 647.016,A -85,B 0,C 180,E1 7002.167,E2 7002.167} C_VEL
LIN {X 0,Y 476.269,Z 670.659,A -85,B 0,C 180,E1 7004.018,E2 7004.018} C_VEL
LIN {X 0,Y 475.507,Z 690.59,A -85,B 0,C 180,E1 7006.46,E2 7006.46} C_VEL
LIN {X 0,Y 475.034,Z 705.708,A -85,B 0,C 180,E1 7009.389,E2 7009.389} C_VEL
LIN {X 0,Y 474.731,Z 714.845,A -85,B 0,C 180,E1 7012.503,E2 7012.503} C_VEL
LIN {X 0,Y 474.663,Z 717.786,A -85,B 0,C 180,E1 7014.523,E2 7014.523} C_VEL
LIN {X 0,Y 474.665,Z 718.459,A -85,B 0,C 180,E1 7016.35,E2 7016.35} C_VEL
LIN {X 0,Y 474.794,Z 716.092,A -85,B 0,C 180,E1 7019.085,E2 7019.085} C_VEL
LIN {X 0,Y 475.16,Z 707.812,A -85,B 0,C 180,E1 7022.271,E2 7022.271} C_VEL
LIN {X 0,Y 475.706,Z 694.949,A -85,B 0,C 180,E1 7025,E2 7025} C_VEL
LIN {X 0,Y 476.43,Z 676.251,A -85,B 0,C 180,E1 7027.503,E2 7027.503} C_VEL
LIN {X 0,Y 477.076,Z 653.48,A -85,B 0,C 180,E1 7029.44,E2 7029.44} C_VEL
LIN {X 0,Y 477.468,Z 627.022,A -85,B 0,C 180,E1 7030.754,E2 7030.754} C_VEL
LIN {X 0,Y 477.498,Z 592.512,A -85,B 0,C 180,E1 7031.481,E2 7031.481} C_VEL
LIN {X 0,Y 476.863,Z 565.585,A -85,B 0,C 180,E1 7031.939,E2 7031.939} C_VEL
LIN {X 0,Y 473.146,Z 549.53,A -85,B 0,C 180,E1 7032.393,E2 7032.393} C_VEL
LIN {X 0,Y 472.886,Z 549.53,A -85,B 0,C 180,E1 7038.605,E2 7038.605} C_VEL
LIN {X 0,Y 472.712,Z 549.53,A -85,B 0,C 180,E1 7044.514,E2 7044.514} C_VEL
LIN {X 0,Y 472.506,Z 549.53,A -85,B 0,C 180,E1 7050.725,E2 7050.725} C_VEL
LIN {X 0,Y 472.609,Z 549.53,A -85,B 0,C 180,E1 7057.343,E2 7057.343} C_VEL
LIN {X 0,Y 472.421,Z 549.53,A -85,B 0,C 180,E1 7063.592,E2 7063.592} C_VEL
LIN {X 0,Y 472.426,Z 549.53,A -85,B 0,C 180,E1 7067.694,E2 7067.694} C_VEL
LIN {X 0,Y 468.455,Z 549.53,A -85,B 0,C 180,E1 7068.453,E2 7068.453} C_VEL
LIN {X 0,Y 464.5,Z 549.53,A -85,B 0,C 180,E1 7069.224,E2 7069.224} C_VEL
LIN {X 0,Y 464.608,Z 549.75,A -85,B 0,C 180,E1 7070.193,E2 7070.193} C_VEL
LIN {X 0,Y 481.222,Z 589.691,A -85,B 0,C 180,E1 7072.5,E2 7072.5} C_VEL
LIN {X 0,Y 487.593,Z 598.553,A -85,B 0,C 180,E1 7073.187,E2 7073.187} C_VEL
LIN {X 0,Y 485.329,Z 642.622,A -85,B 0,C 180,E1 7074.403,E2 7074.403} C_VEL
LIN {X 0,Y 482.291,Z 683.272,A -85,B 0,C 180,E1 7076.277,E2 7076.277} C_VEL
LIN {X 0,Y 478.649,Z 721.142,A -85,B 0,C 180,E1 7078.809,E2 7078.809} C_VEL
LIN {X 0,Y 474.957,Z 755.715,A -85,B 0,C 180,E1 7081.986,E2 7081.986} C_VEL
LIN {X 0,Y 471.677,Z 783.284,A -85,B 0,C 180,E1 7085.421,E2 7085.421} C_VEL
LIN {X 0,Y 468.749,Z 809.169,A -85,B 0,C 180,E1 7089.75,E2 7089.75} C_VEL
LIN {X 0,Y 466.998,Z 828.297,A -85,B 0,C 180,E1 7094.056,E2 7094.056} C_VEL
LIN {X 0,Y 466.096,Z 843.319,A -85,B 0,C 180,E1 7098.797,E2 7098.797} C_VEL
LIN {X 0,Y 465.744,Z 852.735,A -85,B 0,C 180,E1 7103.488,E2 7103.488} C_VEL
LIN {X 0,Y 465.611,Z 857.109,A -85,B 0,C 180,E1 7108.142,E2 7108.142} C_VEL
LIN {X 0,Y 465.686,Z 857.109,A -85,B 0,C 180,E1 7111.857,E2 7111.857} C_VEL
LIN {X 0,Y 465.733,Z 852.737,A -85,B 0,C 180,E1 7116.512,E2 7116.512} C_VEL
LIN {X 0,Y 466.005,Z 843.321,A -85,B 0,C 180,E1 7121.204,E2 7121.204} C_VEL
LIN {X 0,Y 467.081,Z 828.3,A -85,B 0,C 180,E1 7125.94,E2 7125.94} C_VEL
LIN {X 0,Y 468.929,Z 807.914,A -85,B 0,C 180,E1 7130.487,E2 7130.487} C_VEL
LIN {X 0,Y 471.926,Z 781.597,A -85,B 0,C 180,E1 7134.817,E2 7134.817} C_VEL
LIN {X 0,Y 475.037,Z 754.749,A -85,B 0,C 180,E1 7138.12,E2 7138.12} C_VEL
LIN {X 0,Y 478.746,Z 720.197,A -85,B 0,C 180,E1 7141.275,E2 7141.275} C_VEL
LIN {X 0,Y 482.414,Z 682.047,A -85,B 0,C 180,E1 7143.808,E2 7143.808} C_VEL
LIN {X 0,Y 485.512,Z 640.378,A -85,B 0,C 180,E1 7145.697,E2 7145.697} C_VEL
LIN {X 0,Y 487.451,Z 597.842,A -85,B 0,C 180,E1 7146.863,E2 7146.863} C_VEL
LIN {X 0,Y 476.504,Z 578.921,A -85,B 0,C 180,E1 7148.122,E2 7148.122} C_VEL
LIN {X 0,Y 464.687,Z 549.53,A -85,B 0,C 180,E1 7149.78,E2 7149.78} C_VEL
LIN {X 0,Y 464.572,Z 549.53,A -85,B 0,C 180,E1 7155.616,E2 7155.616} C_VEL
LIN {X 0,Y 464.636,Z 549.53,A -85,B 0,C 180,E1 7161.903,E2 7161.903} C_VEL
LIN {X 0,Y 464.61,Z 549.53,A -85,B 0,C 180,E1 7168.695,E2 7168.695} C_VEL
LIN {X 0,Y 464.933,Z 549.53,A -85,B 0,C 180,E1 7175.772,E2 7175.772} C_VEL
LIN {X 0,Y 470.689,Z 575.732,A -85,B 0,C 180,E1 7176.475,E2 7176.475} C_VEL
LIN {X 0,Y 470.773,Z 611.325,A -85,B 0,C 180,E1 7177.261,E2 7177.261} C_VEL
LIN {X 0,Y 470.297,Z 639.717,A -85,B 0,C 180,E1 7178.631,E2 7178.631} C_VEL
LIN {X 0,Y 469.458,Z 664.866,A -85,B 0,C 180,E1 7180.645,E2 7180.645} C_VEL
LIN {X 0,Y 468.571,Z 685.549,A -85,B 0,C 180,E1 7183.156,E2 7183.156} C_VEL
LIN {X 0,Y 467.714,Z 701.946,A -85,B 0,C 180,E1 7186.173,E2 7186.173} C_VEL
LIN {X 0,Y 467.209,Z 712.782,A -85,B 0,C 180,E1 7189.399,E2 7189.399} C_VEL
LIN {X 0,Y 466.86,Z 718.163,A -85,B 0,C 180,E1 7192.576,E2 7192.576} C_VEL
LIN {X 0,Y 466.86,Z 718.534,A -85,B 0,C 180,E1 7196.298,E2 7196.298} C_VEL
LIN {X 0,Y 466.911,Z 713.859,A -85,B 0,C 180,E1 7199.541,E2 7199.541} C_VEL
LIN {X 0,Y 467.227,Z 704.106,A -85,B 0,C 180,E1 7202.781,E2 7202.781} C_VEL
LIN {X 0,Y 467.966,Z 688.001,A -85,B 0,C 180,E1 7206.02,E2 7206.02} C_VEL
LIN {X 0,Y 468.917,Z 667.026,A -85,B 0,C 180,E1 7208.797,E2 7208.797} C_VEL
LIN {X 0,Y 469.897,Z 642.123,A -85,B 0,C 180,E1 7210.997,E2 7210.997} C_VEL
LIN {X 0,Y 470.727,Z 614.918,A -85,B 0,C 180,E1 7212.523,E2 7212.523} C_VEL
LIN {X 0,Y 471.153,Z 586.678,A -85,B 0,C 180,E1 7213.381,E2 7213.381} C_VEL
LIN {X 0,Y 469.955,Z 568.546,A -85,B 0,C 180,E1 7213.731,E2 7213.731} C_VEL
LIN {X 0,Y 465.262,Z 549.53,A -85,B 0,C 180,E1 7214.303,E2 7214.303} C_VEL
LIN {X 0,Y 464.977,Z 549.53,A -85,B 0,C 180,E1 7220.92,E2 7220.92} C_VEL
LIN {X 0,Y 464.756,Z 549.53,A -85,B 0,C 180,E1 7227.042,E2 7227.042} C_VEL
LIN {X 0,Y 464.616,Z 549.53,A -85,B 0,C 180,E1 7233.519,E2 7233.519} C_VEL
LIN {X 0,Y 464.457,Z 549.53,A -85,B 0,C 180,E1 7240.532,E2 7240.532} C_VEL
LIN {X 0,Y 464.575,Z 549.53,A -85,B 0,C 180,E1 7246.986,E2 7246.986} C_VEL
LIN {X 0,Y 464.571,Z 549.53,A -85,B 0,C 180,E1 7251.887,E2 7251.887} C_VEL
LIN {X 0,Y 464.54,Z 549.53,A -85,B 0,C 180,E1 7257.636,E2 7257.636} C_VEL
LIN {X 0,Y 464.726,Z 549.53,A -85,B 0,C 180,E1 7259.603,E2 7259.603} C_VEL
LIN {X 0,Y 481.142,Z 591.814,A -85,B 0,C 180,E1 7262.048,E2 7262.048} C_VEL
LIN {X 0,Y 478.846,Z 627.388,A -85,B 0,C 180,E1 7263.642,E2 7263.642} C_VEL
LIN {X 0,Y 475.913,Z 661.199,A -85,B 0,C 180,E1 7265.928,E2 7265.928} C_VEL
LIN {X 0,Y 472.875,Z 692.027,A -85,B 0,C 180,E1 7268.836,E2 7268.836} C_VEL
LIN {X 0,Y 470.07,Z 718.298,A -85,B 0,C 180,E1 7272.242,E2 7272.242} C_VEL
LIN {X 0,Y 467.928,Z 739.883,A -85,B 0,C 180,E1 7276.031,E2 7276.031} C_VEL
LIN {X 0,Y 466.594,Z 757.326,A -85,B 0,C 180,E1 7280.305,E2 7280.305} C_VEL
LIN {X 0,Y 465.916,Z 768.565,A -85,B 0,C 180,E1 7284.424,E2 7284.424} C_VEL
LIN {X 0,Y 465.744,Z 774.728,A -85,B 0,C 180,E1 7288.143,E2 7288.143} C_VEL
LIN {X 0,Y 465.639,Z 777.432,A -85,B 0,C 180,E1 7291.858,E2 7291.858} C_VEL
LIN {X 0,Y 465.613,Z 776.742,A -85,B 0,C 180,E1 7295.58,E2 7295.58} C_VEL
LIN {X 0,Y 465.787,Z 772.607,A -85,B 0,C 180,E1 7299.324,E2 7299.324} C_VEL
LIN {X 0,Y 466.249,Z 762.791,A -85,B 0,C 180,E1 7303.824,E2 7303.824} C_VEL
LIN {X 0,Y 467.389,Z 746.821,A -85,B 0,C 180,E1 7308.365,E2 7308.365} C_VEL
LIN {X 0,Y 469.293,Z 725.995,A -85,B 0,C 180,E1 7312.45,E2 7312.45} C_VEL
LIN {X 0,Y 471.988,Z 700.742,A -85,B 0,C 180,E1 7316.06,E2 7316.06} C_VEL
LIN {X 0,Y 474.997,Z 670.601,A -85,B 0,C 180,E1 7319.192,E2 7319.192} C_VEL
LIN {X 0,Y 478.091,Z 636.465,A -85,B 0,C 180,E1 7321.733,E2 7321.733} C_VEL
LIN {X 0,Y 480.554,Z 600.038,A -85,B 0,C 180,E1 7323.555,E2 7323.555} C_VEL
LIN {X 0,Y 480.307,Z 589.264,A -85,B 0,C 180,E1 7324.007,E2 7324.007} C_VEL
LIN {X 0,Y 465.578,Z 552.754,A -85,B 0,C 180,E1 7326.211,E2 7326.211} C_VEL
LIN {X 0,Y 464.88,Z 549.53,A -85,B 0,C 180,E1 7326.366,E2 7326.366} C_VEL
LIN {X 0,Y 464.552,Z 549.53,A -85,B 0,C 180,E1 7333.018,E2 7333.018} C_VEL
LIN {X 0,Y 464.569,Z 549.53,A -85,B 0,C 180,E1 7339.479,E2 7339.479} C_VEL
LIN {X 0,Y 464.818,Z 549.53,A -85,B 0,C 180,E1 7344.263,E2 7344.263} C_VEL
LIN {X 0,Y 464.709,Z 549.53,A -85,B 0,C 180,E1 7350.846,E2 7350.846} C_VEL
LIN {X 0,Y 464.737,Z 549.53,A -85,B 0,C 180,E1 7357.063,E2 7357.063} C_VEL
LIN {X 0,Y 464.902,Z 549.53,A -85,B 0,C 180,E1 7359.285,E2 7359.285} C_VEL
LIN {X 0,Y 469.878,Z 576.15,A -85,B 0,C 180,E1 7359.902,E2 7359.902} C_VEL
LIN {X 0,Y 469.761,Z 622.745,A -85,B 0,C 180,E1 7360.799,E2 7360.799} C_VEL
LIN {X 0,Y 469.265,Z 648.555,A -85,B 0,C 180,E1 7362.008,E2 7362.008} C_VEL
LIN {X 0,Y 468.56,Z 671.895,A -85,B 0,C 180,E1 7363.868,E2 7363.868} C_VEL
LIN {X 0,Y 467.773,Z 691.601,A -85,B 0,C 180,E1 7366.308,E2 7366.308} C_VEL
LIN {X 0,Y 467.319,Z 706.101,A -85,B 0,C 180,E1 7369.101,E2 7369.101} C_VEL
LIN {X 0,Y 466.975,Z 715.397,A -85,B 0,C 180,E1 7372.102,E2 7372.102} C_VEL
LIN {X 0,Y 466.889,Z 719,A -85,B 0,C 180,E1 7374.431,E2 7374.431} C_VEL
LIN {X 0,Y 466.889,Z 719.783,A -85,B 0,C 180,E1 7376.289,E2 7376.289} C_VEL
LIN {X 0,Y 467.036,Z 717.538,A -85,B 0,C 180,E1 7379.07,E2 7379.07} C_VEL
LIN {X 0,Y 467.427,Z 709.379,A -85,B 0,C 180,E1 7382.309,E2 7382.309} C_VEL
LIN {X 0,Y 468.027,Z 696.617,A -85,B 0,C 180,E1 7385.083,E2 7385.083} C_VEL
LIN {X 0,Y 468.771,Z 678.06,A -85,B 0,C 180,E1 7387.626,E2 7387.626} C_VEL
LIN {X 0,Y 469.455,Z 655.498,A -85,B 0,C 180,E1 7389.595,E2 7389.595} C_VEL
LIN {X 0,Y 469.843,Z 629.526,A -85,B 0,C 180,E1 7390.931,E2 7390.931} C_VEL
LIN {X 0,Y 469.858,Z 596.2,A -85,B 0,C 180,E1 7391.671,E2 7391.671} C_VEL
LIN {X 0,Y 469.343,Z 567.064,A -85,B 0,C 180,E1 7392.173,E2 7392.173} C_VEL
LIN {X 0,Y 465.218,Z 549.53,A -85,B 0,C 180,E1 7392.647,E2 7392.647} C_VEL
LIN {X 0,Y 464.935,Z 549.53,A -85,B 0,C 180,E1 7398.935,E2 7398.935} C_VEL
LIN {X 0,Y 464.742,Z 549.53,A -85,B 0,C 180,E1 7404.963,E2 7404.963} C_VEL
LIN {X 0,Y 464.532,Z 549.53,A -85,B 0,C 180,E1 7411.311,E2 7411.311} C_VEL
LIN {X 0,Y 464.598,Z 549.53,A -85,B 0,C 180,E1 7418.101,E2 7418.101} C_VEL
LIN {X 0,Y 464.551,Z 549.53,A -85,B 0,C 180,E1 7424.38,E2 7424.38} C_VEL
LIN {X 0,Y 464.5,Z 549.53,A -85,B 0,C 180,E1 7429.224,E2 7429.224} C_VEL
LIN {X 0,Y 464.764,Z 552.619,A -85,B 0,C 180,E1 7429.988,E2 7429.988} C_VEL
LIN {X 0,Y 465.686,Z 562.196,A -85,B 0,C 180,E1 7430.626,E2 7430.626} C_VEL
LIN {X 0,Y 468.958,Z 580.155,A -85,B 0,C 180,E1 7431.266,E2 7431.266} C_VEL
LIN {X 0,Y 479.122,Z 599.757,A -85,B 0,C 180,E1 7432.543,E2 7432.543} C_VEL
LIN {X 0,Y 480.873,Z 602.07,A -85,B 0,C 180,E1 7432.742,E2 7432.742} C_VEL
LIN {X 0,Y 478.338,Z 645.161,A -85,B 0,C 180,E1 7434.011,E2 7434.011} C_VEL
LIN {X 0,Y 475.063,Z 685.469,A -85,B 0,C 180,E1 7435.95,E2 7435.95} C_VEL
LIN {X 0,Y 471.134,Z 723.966,A -85,B 0,C 180,E1 7438.629,E2 7438.629} C_VEL
LIN {X 0,Y 467.162,Z 758.488,A -85,B 0,C 180,E1 7441.936,E2 7441.936} C_VEL
LIN {X 0,Y 463.612,Z 788.564,A -85,B 0,C 180,E1 7445.815,E2 7445.815} C_VEL
LIN {X 0,Y 460.802,Z 812.767,A -85,B 0,C 180,E1 7450.135,E2 7450.135} C_VEL
LIN {X 0,Y 459.004,Z 831.785,A -85,B 0,C 180,E1 7454.749,E2 7454.749} C_VEL
LIN {X 0,Y 458.184,Z 845.62,A -85,B 0,C 180,E1 7459.562,E2 7459.562} C_VEL
LIN {X 0,Y 457.754,Z 853.994,A -85,B 0,C 180,E1 7464.323,E2 7464.323} C_VEL
LIN {X 0,Y 457.706,Z 857.108,A -85,B 0,C 180,E1 7468.11,E2 7468.11} C_VEL
LIN {X 0,Y 457.78,Z 857.108,A -85,B 0,C 180,E1 7471.889,E2 7471.889} C_VEL
LIN {X 0,Y 457.842,Z 852.736,A -85,B 0,C 180,E1 7476.625,E2 7476.625} C_VEL
LIN {X 0,Y 458.176,Z 843.32,A -85,B 0,C 180,E1 7481.398,E2 7481.398} C_VEL
LIN {X 0,Y 459.327,Z 828.299,A -85,B 0,C 180,E1 7486.217,E2 7486.217} C_VEL
LIN {X 0,Y 461.325,Z 807.913,A -85,B 0,C 180,E1 7490.84,E2 7490.84} C_VEL
LIN {X 0,Y 464.13,Z 784.419,A -85,B 0,C 180,E1 7494.792,E2 7494.792} C_VEL
LIN {X 0,Y 467.826,Z 752.926,A -85,B 0,C 180,E1 7498.676,E2 7498.676} C_VEL
LIN {X 0,Y 471.774,Z 718.119,A -85,B 0,C 180,E1 7501.853,E2 7501.853} C_VEL
LIN {X 0,Y 475.564,Z 680.134,A -85,B 0,C 180,E1 7504.372,E2 7504.372} C_VEL
LIN {X 0,Y 478.821,Z 639.299,A -85,B 0,C 180,E1 7506.224,E2 7506.224} C_VEL
LIN {X 0,Y 480.535,Z 600.941,A -85,B 0,C 180,E1 7507.334,E2 7507.334} C_VEL
LIN {X 0,Y 469.557,Z 580.077,A -85,B 0,C 180,E1 7508.702,E2 7508.702} C_VEL
LIN {X 0,Y 456.687,Z 549.53,A -85,B 0,C 180,E1 7510.544,E2 7510.544} C_VEL
LIN {X 0,Y 456.7,Z 549.53,A -85,B 0,C 180,E1 7516.635,E2 7516.635} C_VEL
LIN {X 0,Y 456.691,Z 549.53,A -85,B 0,C 180,E1 7522.476,E2 7522.476} C_VEL
LIN {X 0,Y 456.664,Z 549.53,A -85,B 0,C 180,E1 7529.231,E2 7529.231} C_VEL
LIN {X 0,Y 457.043,Z 549.53,A -85,B 0,C 180,E1 7535.457,E2 7535.457} C_VEL
LIN {X 0,Y 463.182,Z 578.26,A -85,B 0,C 180,E1 7536.235,E2 7536.235} C_VEL
LIN {X 0,Y 463.223,Z 613.234,A -85,B 0,C 180,E1 7537.03,E2 7537.03} C_VEL
LIN {X 0,Y 462.77,Z 640.713,A -85,B 0,C 180,E1 7538.373,E2 7538.373} C_VEL
LIN {X 0,Y 461.877,Z 666.258,A -85,B 0,C 180,E1 7540.439,E2 7540.439} C_VEL
LIN {X 0,Y 460.963,Z 686.235,A -85,B 0,C 180,E1 7542.869,E2 7542.869} C_VEL
LIN {X 0,Y 460.1,Z 702.034,A -85,B 0,C 180,E1 7545.726,E2 7545.726} C_VEL
LIN {X 0,Y 459.49,Z 713.697,A -85,B 0,C 180,E1 7549.12,E2 7549.12} C_VEL
LIN {X 0,Y 459.099,Z 719.466,A -85,B 0,C 180,E1 7552.449,E2 7552.449} C_VEL
LIN {X 0,Y 459.053,Z 720.481,A -85,B 0,C 180,E1 7554.345,E2 7554.345} C_VEL
LIN {X 0,Y 459.144,Z 717.858,A -85,B 0,C 180,E1 7558.121,E2 7558.121} C_VEL
LIN {X 0,Y 459.333,Z 710.374,A -85,B 0,C 180,E1 7561.416,E2 7561.416} C_VEL
LIN {X 0,Y 459.864,Z 697.171,A -85,B 0,C 180,E1 7564.71,E2 7564.71} C_VEL
LIN {X 0,Y 460.671,Z 679.946,A -85,B 0,C 180,E1 7567.533,E2 7567.533} C_VEL
LIN {X 0,Y 461.709,Z 657.87,A -85,B 0,C 180,E1 7570.003,E2 7570.003} C_VEL
LIN {X 0,Y 462.656,Z 631.848,A -85,B 0,C 180,E1 7571.941,E2 7571.941} C_VEL
LIN {X 0,Y 463.305,Z 602.956,A -85,B 0,C 180,E1 7573.238,E2 7573.238} C_VEL
LIN {X 0,Y 462.731,Z 571.459,A -85,B 0,C 180,E1 7573.934,E2 7573.934} C_VEL
LIN {X 0,Y 457.329,Z 549.53,A -85,B 0,C 180,E1 7574.59,E2 7574.59} C_VEL
LIN {X 0,Y 457.018,Z 549.53,A -85,B 0,C 180,E1 7581.302,E2 7581.302} C_VEL
LIN {X 0,Y 456.823,Z 549.53,A -85,B 0,C 180,E1 7587.551,E2 7587.551} C_VEL
LIN {X 0,Y 456.626,Z 549.53,A -85,B 0,C 180,E1 7594.284,E2 7594.284} C_VEL
LIN {X 0,Y 456.574,Z 549.53,A -85,B 0,C 180,E1 7600.514,E2 7600.514} C_VEL
LIN {X 0,Y 456.643,Z 549.53,A -85,B 0,C 180,E1 7606.643,E2 7606.643} C_VEL
LIN {X 0,Y 456.636,Z 549.53,A -85,B 0,C 180,E1 7612.485,E2 7612.485} C_VEL
LIN {X 0,Y 456.718,Z 549.53,A -85,B 0,C 180,E1 7618.93,E2 7618.93} C_VEL
LIN {X 0,Y 474.103,Z 593.094,A -85,B 0,C 180,E1 7621.61,E2 7621.61} C_VEL
LIN {X 0,Y 471.671,Z 629.404,A -85,B 0,C 180,E1 7623.299,E2 7623.299} C_VEL
LIN {X 0,Y 468.592,Z 662.944,A -85,B 0,C 180,E1 7625.629,E2 7625.629} C_VEL
LIN {X 0,Y 465.379,Z 693.718,A -85,B 0,C 180,E1 7628.609,E2 7628.609} C_VEL
LIN {X 0,Y 462.385,Z 720.534,A -85,B 0,C 180,E1 7632.183,E2 7632.183} C_VEL
LIN {X 0,Y 459.998,Z 743.167,A -85,B 0,C 180,E1 7636.325,E2 7636.325} C_VEL
LIN {X 0,Y 458.645,Z 760.135,A -85,B 0,C 180,E1 7640.798,E2 7640.798} C_VEL
LIN {X 0,Y 458.1,Z 771.209,A -85,B 0,C 180,E1 7645.276,E2 7645.276} C_VEL
LIN {X 0,Y 457.943,Z 777.274,A -85,B 0,C 180,E1 7650,E2 7650} C_VEL
LIN {X 0,Y 457.801,Z 778.216,A -85,B 0,C 180,E1 7653.781,E2 7653.781} C_VEL
LIN {X 0,Y 457.902,Z 774.531,A -85,B 0,C 180,E1 7658.609,E2 7658.609} C_VEL
LIN {X 0,Y 458.316,Z 765.233,A -85,B 0,C 180,E1 7663.327,E2 7663.327} C_VEL
LIN {X 0,Y 459.435,Z 751.031,A -85,B 0,C 180,E1 7667.714,E2 7667.714} C_VEL
LIN {X 0,Y 461.271,Z 731.749,A -85,B 0,C 180,E1 7671.85,E2 7671.85} C_VEL
LIN {X 0,Y 463.933,Z 706.701,A -85,B 0,C 180,E1 7675.708,E2 7675.708} C_VEL
LIN {X 0,Y 467.082,Z 677.512,A -85,B 0,C 180,E1 7678.991,E2 7678.991} C_VEL
LIN {X 0,Y 470.327,Z 644.315,A -85,B 0,C 180,E1 7681.676,E2 7681.676} C_VEL
LIN {X 0,Y 473.222,Z 608.178,A -85,B 0,C 180,E1 7683.703,E2 7683.703} C_VEL
LIN {X 0,Y 473.442,Z 591.658,A -85,B 0,C 180,E1 7684.415,E2 7684.415} C_VEL
LIN {X 0,Y 459.687,Z 556.894,A -85,B 0,C 180,E1 7686.612,E2 7686.612} C_VEL
LIN {X 0,Y 456.881,Z 549.53,A -85,B 0,C 180,E1 7687.111,E2 7687.111} C_VEL
LIN {X 0,Y 456.602,Z 549.53,A -85,B 0,C 180,E1 7693.956,E2 7693.956} C_VEL
LIN {X 0,Y 456.683,Z 549.53,A -85,B 0,C 180,E1 7699.471,E2 7699.471} C_VEL
LIN {X 0,Y 456.827,Z 549.53,A -85,B 0,C 180,E1 7705.831,E2 7705.831} C_VEL
LIN {X 0,Y 456.792,Z 549.53,A -85,B 0,C 180,E1 7712.447,E2 7712.447} C_VEL
LIN {X 0,Y 456.953,Z 549.53,A -85,B 0,C 180,E1 7719.004,E2 7719.004} C_VEL
LIN {X 0,Y 462.121,Z 575.642,A -85,B 0,C 180,E1 7719.644,E2 7719.644} C_VEL
LIN {X 0,Y 462.088,Z 624.162,A -85,B 0,C 180,E1 7720.601,E2 7720.601} C_VEL
LIN {X 0,Y 461.56,Z 650.487,A -85,B 0,C 180,E1 7721.871,E2 7721.871} C_VEL
LIN {X 0,Y 460.835,Z 674.272,A -85,B 0,C 180,E1 7723.835,E2 7723.835} C_VEL
LIN {X 0,Y 459.976,Z 693.814,A -85,B 0,C 180,E1 7726.346,E2 7726.346} C_VEL
LIN {X 0,Y 459.534,Z 707.921,A -85,B 0,C 180,E1 7729.16,E2 7729.16} C_VEL
LIN {X 0,Y 459.202,Z 717.529,A -85,B 0,C 180,E1 7732.478,E2 7732.478} C_VEL
LIN {X 0,Y 459.122,Z 720.211,A -85,B 0,C 180,E1 7734.337,E2 7734.337} C_VEL
LIN {X 0,Y 459.123,Z 721.097,A -85,B 0,C 180,E1 7736.227,E2 7736.227} C_VEL
LIN {X 0,Y 459.253,Z 718.984,A -85,B 0,C 180,E1 7739.054,E2 7739.054} C_VEL
LIN {X 0,Y 459.684,Z 710.965,A -85,B 0,C 180,E1 7742.347,E2 7742.347} C_VEL
LIN {X 0,Y 460.327,Z 698.338,A -85,B 0,C 180,E1 7745.168,E2 7745.168} C_VEL
LIN {X 0,Y 461.126,Z 679.902,A -85,B 0,C 180,E1 7747.754,E2 7747.754} C_VEL
LIN {X 0,Y 461.839,Z 657.504,A -85,B 0,C 180,E1 7749.754,E2 7749.754} C_VEL
LIN {X 0,Y 462.244,Z 631.975,A -85,B 0,C 180,E1 7751.113,E2 7751.113} C_VEL
LIN {X 0,Y 462.237,Z 599.882,A -85,B 0,C 180,E1 7751.872,E2 7751.872} C_VEL
LIN {X 0,Y 461.56,Z 567.277,A -85,B 0,C 180,E1 7752.458,E2 7752.458} C_VEL
LIN {X 0,Y 457.277,Z 549.53,A -85,B 0,C 180,E1 7752.982,E2 7752.982} C_VEL
LIN {X 0,Y 457.012,Z 549.53,A -85,B 0,C 180,E1 7759.276,E2 7759.276} C_VEL
LIN {X 0,Y 456.773,Z 549.53,A -85,B 0,C 180,E1 7765.43,E2 7765.43} C_VEL
LIN {X 0,Y 456.608,Z 549.53,A -85,B 0,C 180,E1 7771.918,E2 7771.918} C_VEL
LIN {X 0,Y 456.686,Z 549.53,A -85,B 0,C 180,E1 7778.884,E2 7778.884} C_VEL
LIN {X 0,Y 456.664,Z 549.53,A -85,B 0,C 180,E1 7783.937,E2 7783.937} C_VEL
LIN {X 0,Y 456.633,Z 549.53,A -85,B 0,C 180,E1 7789.464,E2 7789.464} C_VEL
